LIN {X -0.161,Y -632.553,Z 539.342,A 0.000,B 0.000,C 90.000,E1 97.587} C_DIS
LIN {X 0.137,Y -636.870,Z 539.336,A 0.000,B 0.000,C 90.000,E1 96.549} C_DIS
LIN {X 0.117,Y -640.044,Z 539.332,A 0.000,B 0.000,C 90.000,E1 95.796} C_DIS
LIN {X -0.184,Y -643.748,Z 539.327,A 0.000,B 0.000,C 90.000,E1 94.821} C_DIS
LIN {X -0.199,Y -646.261,Z 539.323,A 0.000,B 0.000,C 90.000,E1 94.073} C_DIS
LIN {X -0.191,Y -648.527,Z 539.318,A 0.000,B 0.000,C 90.000,E1 93.326} C_DIS
LIN {X -0.164,Y -650.528,Z 539.314,A 0.000,B 0.000,C 90.000,E1 92.579} C_DIS
LIN {X -0.144,Y -652.163,Z 539.310,A 0.000,B 0.000,C 90.000,E1 91.835} C_DIS
LIN {X -0.091,Y -653.365,Z 539.306,A 0.000,B 0.000,C 90.000,E1 91.088} C_DIS
LIN {X 0.160,Y -654.029,Z 539.303,A 0.000,B 0.000,C 90.000,E1 90.573} C_DIS
LIN {X -0.239,Y -654.516,Z 539.301,A 0.000,B 0.000,C 90.000,E1 90.115} C_DIS
LIN {X -0.177,Y -654.885,Z 539.296,A 0.000,B 0.000,C 90.000,E1 89.370} C_DIS
LIN {X 0.085,Y -654.983,Z 539.294,A 0.000,B 0.000,C 90.000,E1 88.854} C_DIS
LIN {X 0.168,Y -654.825,Z 539.290,A 0.000,B 0.000,C 90.000,E1 88.108} C_DIS
LIN {X -0.226,Y -654.541,Z 539.287,A 0.000,B 0.000,C 90.000,E1 87.650} C_DIS
LIN {X -0.173,Y -653.859,Z 539.283,A 0.000,B 0.000,C 90.000,E1 86.906} C_DIS
LIN {X -0.257,Y -652.473,Z 539.277,A 0.000,B 0.000,C 90.000,E1 85.927} C_DIS
LIN {X 0.186,Y -652.109,Z 539.276,A 0.000,B 0.000,C 90.000,E1 85.641} C_DIS
LIN {X -0.127,Y -649.508,Z 539.269,A 0.000,B 0.000,C 90.000,E1 84.432} C_DIS
LIN {X 0.138,Y -648.367,Z 539.266,A 0.000,B 0.000,C 90.000,E1 83.913} C_DIS
LIN {X 0.000,Y -645.573,Z 539.261,A 0.000,B 0.000,C 90.000,E1 82.932} C_DIS
LIN {X 0.237,Y -643.951,Z 539.258,A 0.000,B 0.000,C 90.000,E1 82.413} C_DIS
LIN {X 0.034,Y -640.529,Z 539.252,A 0.000,B 0.000,C 90.000,E1 81.432} C_DIS
LIN {X 0.227,Y -638.679,Z 539.250,A 0.000,B 0.000,C 90.000,E1 80.914} C_DIS
LIN {X 0.333,Y -635.655,Z 539.245,A 0.000,B 0.000,C 90.000,E1 80.151} C_DIS
LIN {X -0.136,Y -633.425,Z 539.243,A 0.000,B 0.000,C 90.000,E1 79.690} C_DIS
LIN {X -0.226,Y -629.355,Z 539.238,A 0.000,B 0.000,C 90.000,E1 78.814} C_DIS
LIN {X -0.190,Y -625.693,Z 539.234,A 0.000,B 0.000,C 90.000,E1 78.049} C_DIS
LIN {X -0.215,Y -619.808,Z 539.227,A 0.000,B 0.000,C 90.000,E1 76.937} C_DIS
LIN {X -0.057,Y -616.886,Z 539.224,A 0.000,B 0.000,C 90.000,E1 76.408} C_DIS
LIN {X -0.161,Y -612.053,Z 539.220,A 0.000,B 0.000,C 90.000,E1 75.644} C_DIS
LIN {X 0.217,Y -605.780,Z 539.215,A 0.000,B 0.000,C 90.000,E1 74.700} C_DIS
LIN {X 0.209,Y -600.730,Z 539.212,A 0.000,B 0.000,C 90.000,E1 74.047} C_DIS
LIN {X -0.187,Y -596.279,Z 539.209,A 0.000,B 0.000,C 90.000,E1 73.559} C_DIS
LIN {X -0.213,Y -590.050,Z 539.205,A 0.000,B 0.000,C 90.000,E1 72.906} C_DIS
LIN {X 0.120,Y -586.238,Z 539.203,A 0.000,B 0.000,C 90.000,E1 72.489} C_DIS
LIN {X 0.255,Y -580.969,Z 539.200,A 0.000,B 0.000,C 90.000,E1 72.000} C_DIS
LIN {X -0.331,Y -573.128,Z 539.197,A 0.000,B 0.000,C 90.000,E1 71.402} C_DIS
LIN {X -0.139,Y -568.567,Z 539.195,A 0.000,B 0.000,C 90.000,E1 71.040} C_DIS
LIN {X 0.221,Y -563.998,Z 539.193,A 0.000,B 0.000,C 90.000,E1 70.678} C_DIS
LIN {X -0.057,Y -557.456,Z 539.191,A 0.000,B 0.000,C 90.000,E1 70.296} C_DIS
LIN {X 0.145,Y -549.435,Z 539.188,A 0.000,B 0.000,C 90.000,E1 69.826} C_DIS
LIN {X -0.129,Y -542.518,Z 539.186,A 0.000,B 0.000,C 90.000,E1 69.518} C_DIS
LIN {X -0.088,Y -535.231,Z 539.185,A 0.000,B 0.000,C 90.000,E1 69.209} C_DIS
LIN {X -0.199,Y -527.996,Z 539.183,A 0.000,B 0.000,C 90.000,E1 68.954} C_DIS
LIN {X -0.211,Y -517.329,Z 539.181,A 0.000,B 0.000,C 90.000,E1 68.592} C_DIS
LIN {X 0.274,Y -504.903,Z 539.179,A 0.000,B 0.000,C 90.000,E1 68.156} C_DIS
LIN {X -0.019,Y -497.455,Z 539.178,A 0.000,B 0.000,C 90.000,E1 67.975} C_DIS
LIN {X 0.175,Y -485.004,Z 539.176,A 0.000,B 0.000,C 90.000,E1 67.614} C_DIS
LIN {X 0.015,Y -465.783,Z 539.173,A 0.000,B 0.000,C 90.000,E1 67.102} C_DIS
LIN {X -0.011,Y -465.706,Z 539.173,A 0.000,B 0.000,C 90.000,E1 67.102} C_DIS
LIN {X -0.282,Y -455.953,Z 539.146,A 0.000,B 0.000,C 90.000,E1 62.231} C_DIS
LIN {X -0.176,Y -455.427,Z 539.144,A 0.000,B 0.000,C 90.000,E1 61.897} C_DIS
LIN {X 0.140,Y -446.089,Z 539.120,A 0.000,B 0.000,C 90.000,E1 57.661} C_DIS
LIN {X 0.017,Y -443.661,Z 539.113,A 0.000,B 0.000,C 90.000,E1 56.373} C_DIS
LIN {X 0.047,Y -443.048,Z 539.112,A 0.000,B 0.000,C 90.000,E1 56.135} C_DIS
LIN {X 0.007,Y -443.048,Z 539.112,A 0.000,B 0.000,C 90.000,E1 56.135} C_DIS
LIN {X 0.110,Y -446.646,Z 539.102,A 0.000,B 0.000,C 90.000,E1 54.402} C_DIS
LIN {X 0.221,Y -449.820,Z 539.093,A 0.000,B 0.000,C 90.000,E1 52.763} C_DIS
LIN {X 0.040,Y -452.125,Z 539.086,A 0.000,B 0.000,C 90.000,E1 51.492} C_DIS
LIN {X 0.099,Y -453.720,Z 539.081,A 0.000,B 0.000,C 90.000,E1 50.517} C_DIS
LIN {X 0.196,Y -455.801,Z 539.074,A 0.000,B 0.000,C 90.000,E1 49.218} C_DIS
LIN {X 0.025,Y -457.655,Z 539.066,A 0.000,B 0.000,C 90.000,E1 47.957} C_DIS
LIN {X -0.158,Y -459.271,Z 539.059,A 0.000,B 0.000,C 90.000,E1 46.701} C_DIS
LIN {X 0.003,Y -460.455,Z 539.052,A 0.000,B 0.000,C 90.000,E1 45.405} C_DIS
LIN {X 0.140,Y -461.157,Z 539.047,A 0.000,B 0.000,C 90.000,E1 44.433} C_DIS
LIN {X -0.036,Y -461.732,Z 539.042,A 0.000,B 0.000,C 90.000,E1 43.500} C_DIS
LIN {X 0.160,Y -462.205,Z 539.035,A 0.000,B 0.000,C 90.000,E1 42.204} C_DIS
LIN {X 0.083,Y -462.454,Z 539.028,A 0.000,B 0.000,C 90.000,E1 40.943} C_DIS
LIN {X -0.039,Y -462.485,Z 539.021,A 0.000,B 0.000,C 90.000,E1 39.688} C_DIS
LIN {X 0.248,Y -462.250,Z 539.013,A 0.000,B 0.000,C 90.000,E1 38.382} C_DIS
LIN {X 0.141,Y -461.964,Z 539.008,A 0.000,B 0.000,C 90.000,E1 37.443} C_DIS
LIN {X -0.104,Y -461.385,Z 538.999,A 0.000,B 0.000,C 90.000,E1 35.884} C_DIS
LIN {X -0.117,Y -460.356,Z 538.987,A 0.000,B 0.000,C 90.000,E1 33.658} C_DIS
LIN {X -0.026,Y -459.616,Z 538.978,A 0.000,B 0.000,C 90.000,E1 32.054} C_DIS
LIN {X -0.055,Y -458.897,Z 538.969,A 0.000,B 0.000,C 90.000,E1 30.463} C_DIS
LIN {X -0.200,Y -457.939,Z 538.959,A 0.000,B 0.000,C 90.000,E1 28.565} C_DIS
LIN {X -0.071,Y -457.170,Z 538.950,A 0.000,B 0.000,C 90.000,E1 26.950} C_DIS
LIN {X 0.032,Y -456.139,Z 538.937,A 0.000,B 0.000,C 90.000,E1 24.695} C_DIS
LIN {X -0.155,Y -455.183,Z 538.923,A 0.000,B 0.000,C 90.000,E1 22.153} C_DIS
LIN {X 0.100,Y -454.615,Z 538.912,A 0.000,B 0.000,C 90.000,E1 20.194} C_DIS
LIN {X 0.012,Y -454.238,Z 538.903,A 0.000,B 0.000,C 90.000,E1 18.598} C_DIS
LIN {X 0.057,Y -454.011,Z 538.894,A 0.000,B 0.000,C 90.000,E1 16.985} C_DIS
LIN {X -0.179,Y -453.989,Z 538.878,A 0.000,B 0.000,C 90.000,E1 14.120} C_DIS
LIN {X -0.102,Y -454.567,Z 538.860,A 0.000,B 0.000,C 90.000,E1 10.894} C_DIS
LIN {X -0.233,Y -455.490,Z 538.846,A 0.000,B 0.000,C 90.000,E1 8.341} C_DIS
LIN {X -0.165,Y -456.606,Z 538.834,A 0.000,B 0.000,C 90.000,E1 6.087} C_DIS
LIN {X 0.061,Y -458.239,Z 538.820,A 0.000,B 0.000,C 90.000,E1 3.498} C_DIS
LIN {X 0.078,Y -459.999,Z 538.807,A 0.000,B 0.000,C 90.000,E1 1.260} C_DIS
LIN {X -0.172,Y -463.198,Z 538.790,A 0.000,B 0.000,C 90.000,E1 358.224} C_DIS
LIN {X -0.016,Y -466.734,Z 538.774,A 0.000,B 0.000,C 90.000,E1 355.355} C_DIS
LIN {X 0.090,Y -469.208,Z 538.764,A 0.000,B 0.000,C 90.000,E1 353.451} C_DIS
LIN {X 0.085,Y -472.158,Z 538.752,A 0.000,B 0.000,C 90.000,E1 351.254} C_DIS
LIN {X 0.220,Y -475.229,Z 538.739,A 0.000,B 0.000,C 90.000,E1 349.050} C_DIS
LIN {X -0.047,Y -479.727,Z 538.724,A 0.000,B 0.000,C 90.000,E1 346.284} C_DIS
LIN {X 0.102,Y -484.216,Z 538.710,A 0.000,B 0.000,C 90.000,E1 343.795} C_DIS
LIN {X 0.036,Y -488.962,Z 538.696,A 0.000,B 0.000,C 90.000,E1 341.348} C_DIS
LIN {X 0.038,Y -492.574,Z 538.686,A 0.000,B 0.000,C 90.000,E1 339.518} C_DIS
LIN {X -0.102,Y -496.765,Z 538.674,A 0.000,B 0.000,C 90.000,E1 337.411} C_DIS
LIN {X -0.204,Y -500.238,Z 538.664,A 0.000,B 0.000,C 90.000,E1 335.613} C_DIS
LIN {X -0.180,Y -502.462,Z 538.658,A 0.000,B 0.000,C 90.000,E1 334.409} C_DIS
LIN {X -0.195,Y -505.759,Z 538.648,A 0.000,B 0.000,C 90.000,E1 332.615} C_DIS
LIN {X 0.096,Y -508.923,Z 538.638,A 0.000,B 0.000,C 90.000,E1 330.795} C_DIS
LIN {X 0.269,Y -512.153,Z 538.628,A 0.000,B 0.000,C 90.000,E1 328.997} C_DIS
LIN {X 0.077,Y -515.372,Z 538.618,A 0.000,B 0.000,C 90.000,E1 327.248} C_DIS
LIN {X -0.135,Y -518.119,Z 538.610,A 0.000,B 0.000,C 90.000,E1 325.801} C_DIS
LIN {X -0.001,Y -520.822,Z 538.602,A 0.000,B 0.000,C 90.000,E1 324.322} C_DIS
LIN {X 0.141,Y -524.009,Z 538.592,A 0.000,B 0.000,C 90.000,E1 322.557} C_DIS
LIN {X 0.251,Y -527.316,Z 538.582,A 0.000,B 0.000,C 90.000,E1 320.803} C_DIS
LIN {X -0.116,Y -533.148,Z 538.566,A 0.000,B 0.000,C 90.000,E1 317.957} C_DIS
LIN {X -0.315,Y -537.519,Z 538.555,A 0.000,B 0.000,C 90.000,E1 315.972} C_DIS
LIN {X -0.022,Y -543.522,Z 538.541,A 0.000,B 0.000,C 90.000,E1 313.380} C_DIS
LIN {X 0.027,Y -546.374,Z 538.535,A 0.000,B 0.000,C 90.000,E1 312.243} C_DIS
LIN {X -0.288,Y -549.138,Z 538.529,A 0.000,B 0.000,C 90.000,E1 311.148} C_DIS
LIN {X 0.213,Y -551.048,Z 538.524,A 0.000,B 0.000,C 90.000,E1 310.253} C_DIS
LIN {X 0.008,Y -554.086,Z 538.516,A 0.000,B 0.000,C 90.000,E1 308.874} C_DIS
LIN {X 0.369,Y -557.334,Z 538.508,A 0.000,B 0.000,C 90.000,E1 307.443} C_DIS
LIN {X -0.248,Y -558.907,Z 538.505,A 0.000,B 0.000,C 90.000,E1 306.950} C_DIS
LIN {X -0.037,Y -559.427,Z 538.504,A 0.000,B 0.000,C 90.000,E1 306.790} C_DIS
LIN {X -0.070,Y -561.428,Z 538.502,A 0.000,B 0.000,C 90.000,E1 306.377} C_DIS
LIN {X 0.026,Y -563.355,Z 538.501,A 0.000,B 0.000,C 90.000,E1 306.091} C_DIS
LIN {X 0.129,Y -565.266,Z 538.499,A 0.000,B 0.000,C 90.000,E1 305.804} C_DIS
LIN {X 0.149,Y -568.092,Z 538.497,A 0.000,B 0.000,C 90.000,E1 305.438} C_DIS
LIN {X 0.008,Y -570.735,Z 538.496,A 0.000,B 0.000,C 90.000,E1 305.185} C_DIS
LIN {X 0.208,Y -572.950,Z 538.494,A 0.000,B 0.000,C 90.000,E1 304.898} C_DIS
LIN {X 0.069,Y -576.395,Z 538.492,A 0.000,B 0.000,C 90.000,E1 304.565} C_DIS
LIN {X -0.134,Y -578.700,Z 538.491,A 0.000,B 0.000,C 90.000,E1 304.326} C_DIS
LIN {X -0.132,Y -585.903,Z 538.487,A 0.000,B 0.000,C 90.000,E1 303.579} C_DIS
LIN {X 0.109,Y -591.873,Z 538.483,A 0.000,B 0.000,C 90.000,E1 302.911} C_DIS
LIN {X -0.130,Y -602.582,Z 538.476,A 0.000,B 0.000,C 90.000,E1 301.750} C_DIS
LIN {X 0.293,Y -609.452,Z 538.472,A 0.000,B 0.000,C 90.000,E1 300.924} C_DIS
LIN {X -0.349,Y -614.898,Z 538.468,A 0.000,B 0.000,C 90.000,E1 300.335} C_DIS
LIN {X -0.098,Y -618.893,Z 538.466,A 0.000,B 0.000,C 90.000,E1 299.795} C_DIS
LIN {X -0.125,Y -622.479,Z 538.463,A 0.000,B 0.000,C 90.000,E1 299.283} C_DIS
LIN {X 0.177,Y -625.745,Z 538.460,A 0.000,B 0.000,C 90.000,E1 298.743} C_DIS
LIN {X 0.192,Y -627.757,Z 538.458,A 0.000,B 0.000,C 90.000,E1 298.359} C_DIS
LIN {X 0.231,Y -629.993,Z 538.455,A 0.000,B 0.000,C 90.000,E1 297.847} C_DIS
LIN {X -0.304,Y -630.974,Z 538.453,A 0.000,B 0.000,C 90.000,E1 297.641} C_DIS
LIN {X -0.277,Y -631.817,Z 538.452,A 0.000,B 0.000,C 90.000,E1 297.385} C_DIS
LIN {X -0.212,Y -633.149,Z 538.449,A 0.000,B 0.000,C 90.000,E1 296.873} C_DIS
LIN {X -0.136,Y -633.784,Z 538.446,A 0.000,B 0.000,C 90.000,E1 296.360} C_DIS
LIN {X -0.096,Y -634.016,Z 538.445,A 0.000,B 0.000,C 90.000,E1 296.104} C_DIS
LIN {X -0.015,Y -633.509,Z 538.442,A 0.000,B 0.000,C 90.000,E1 295.591} C_DIS
LIN {X 0.025,Y -633.147,Z 538.441,A 0.000,B 0.000,C 90.000,E1 295.335} C_DIS
LIN {X 0.063,Y -632.018,Z 538.439,A 0.000,B 0.000,C 90.000,E1 295.079} C_DIS
LIN {X 0.100,Y -631.238,Z 538.438,A 0.000,B 0.000,C 90.000,E1 294.823} C_DIS
LIN {X -0.148,Y -630.640,Z 538.437,A 0.000,B 0.000,C 90.000,E1 294.719} C_DIS
LIN {X -0.116,Y -629.010,Z 538.436,A 0.000,B 0.000,C 90.000,E1 294.463} C_DIS
LIN {X -0.102,Y -628.001,Z 538.435,A 0.000,B 0.000,C 90.000,E1 294.335} C_DIS
LIN {X -0.079,Y -625.339,Z 538.434,A 0.000,B 0.000,C 90.000,E1 294.079} C_DIS
LIN {X -0.049,Y -622.387,Z 538.433,A 0.000,B 0.000,C 90.000,E1 293.898} C_DIS
LIN {X 0.191,Y -620.518,Z 538.432,A 0.000,B 0.000,C 90.000,E1 293.695} C_DIS
LIN {X 0.007,Y -618.872,Z 538.431,A 0.000,B 0.000,C 90.000,E1 293.590} C_DIS
LIN {X 0.043,Y -611.966,Z 538.429,A 0.000,B 0.000,C 90.000,E1 293.206} C_DIS
LIN {X -0.106,Y -602.994,Z 538.427,A 0.000,B 0.000,C 90.000,E1 292.823} C_DIS
LIN {X 0.327,Y -596.063,Z 538.425,A 0.000,B 0.000,C 90.000,E1 292.514} C_DIS
LIN {X -0.216,Y -590.775,Z 538.424,A 0.000,B 0.000,C 90.000,E1 292.386} C_DIS
LIN {X -0.212,Y -583.096,Z 538.423,A 0.000,B 0.000,C 90.000,E1 292.078} C_DIS
LIN {X -0.184,Y -578.414,Z 538.421,A 0.000,B 0.000,C 90.000,E1 291.844} C_DIS
LIN {X 0.056,Y -576.702,Z 538.421,A 0.000,B 0.000,C 90.000,E1 291.716} C_DIS
LIN {X -0.083,Y -574.112,Z 538.420,A 0.000,B 0.000,C 90.000,E1 291.535} C_DIS
LIN {X -0.029,Y -573.253,Z 538.419,A 0.000,B 0.000,C 90.000,E1 291.408} C_DIS
LIN {X 0.063,Y -572.549,Z 538.417,A 0.000,B 0.000,C 90.000,E1 291.099} C_DIS
LIN {X -0.328,Y -572.335,Z 538.413,A 0.000,B 0.000,C 90.000,E1 290.429} C_DIS
LIN {X 0.013,Y -572.469,Z 538.409,A 0.000,B 0.000,C 90.000,E1 289.577} C_DIS
LIN {X -0.200,Y -572.511,Z 538.401,A 0.000,B 0.000,C 90.000,E1 288.236} C_DIS
LIN {X -0.053,Y -572.295,Z 538.394,A 0.000,B 0.000,C 90.000,E1 286.858} C_DIS
LIN {X -0.251,Y -571.983,Z 538.388,A 0.000,B 0.000,C 90.000,E1 285.788} C_DIS
LIN {X 0.068,Y -571.227,Z 538.379,A 0.000,B 0.000,C 90.000,E1 284.120} C_DIS
LIN {X 0.091,Y -570.432,Z 538.369,A 0.000,B 0.000,C 90.000,E1 282.479} C_DIS
LIN {X 0.105,Y -569.643,Z 538.360,A 0.000,B 0.000,C 90.000,E1 280.838} C_DIS
LIN {X 0.283,Y -569.045,Z 538.354,A 0.000,B 0.000,C 90.000,E1 279.726} C_DIS
LIN {X 0.059,Y -568.241,Z 538.345,A 0.000,B 0.000,C 90.000,E1 278.106} C_DIS
LIN {X -0.181,Y -567.557,Z 538.336,A 0.000,B 0.000,C 90.000,E1 276.486} C_DIS
LIN {X -0.209,Y -567.219,Z 538.330,A 0.000,B 0.000,C 90.000,E1 275.391} C_DIS
LIN {X 0.165,Y -566.883,Z 538.325,A 0.000,B 0.000,C 90.000,E1 274.531} C_DIS
LIN {X 0.087,Y -566.382,Z 538.319,A 0.000,B 0.000,C 90.000,E1 273.440} C_DIS
LIN {X 0.248,Y -565.415,Z 538.310,A 0.000,B 0.000,C 90.000,E1 271.776} C_DIS
LIN {X 0.129,Y -564.763,Z 538.304,A 0.000,B 0.000,C 90.000,E1 270.688} C_DIS
LIN {X 0.221,Y -563.529,Z 538.295,A 0.000,B 0.000,C 90.000,E1 269.026} C_DIS
LIN {X 0.196,Y -562.554,Z 538.287,A 0.000,B 0.000,C 90.000,E1 267.650} C_DIS
LIN {X -0.092,Y -561.020,Z 538.275,A 0.000,B 0.000,C 90.000,E1 265.469} C_DIS
LIN {X -0.209,Y -560.118,Z 538.269,A 0.000,B 0.000,C 90.000,E1 264.375} C_DIS
LIN {X -0.197,Y -558.958,Z 538.261,A 0.000,B 0.000,C 90.000,E1 262.989} C_DIS
LIN {X -0.150,Y -557.527,Z 538.252,A 0.000,B 0.000,C 90.000,E1 261.319} C_DIS
LIN {X 0.123,Y -556.936,Z 538.249,A 0.000,B 0.000,C 90.000,E1 260.735} C_DIS
LIN {X -0.134,Y -554.565,Z 538.238,A 0.000,B 0.000,C 90.000,E1 258.814} C_DIS
LIN {X -0.167,Y -553.164,Z 538.232,A 0.000,B 0.000,C 90.000,E1 257.701} C_DIS
LIN {X -0.223,Y -551.701,Z 538.225,A 0.000,B 0.000,C 90.000,E1 256.589} C_DIS
LIN {X -0.173,Y -550.104,Z 538.219,A 0.000,B 0.000,C 90.000,E1 255.463} C_DIS
LIN {X 0.102,Y -547.909,Z 538.211,A 0.000,B 0.000,C 90.000,E1 254.031} C_DIS
LIN {X -0.182,Y -545.529,Z 538.204,A 0.000,B 0.000,C 90.000,E1 252.653} C_DIS
LIN {X -0.062,Y -543.444,Z 538.197,A 0.000,B 0.000,C 90.000,E1 251.511} C_DIS
LIN {X 0.019,Y -541.277,Z 538.191,A 0.000,B 0.000,C 90.000,E1 250.369} C_DIS
LIN {X 0.018,Y -539.529,Z 538.186,A 0.000,B 0.000,C 90.000,E1 249.518} C_DIS
LIN {X -0.069,Y -536.536,Z 538.178,A 0.000,B 0.000,C 90.000,E1 248.103} C_DIS
LIN {X 0.282,Y -533.977,Z 538.172,A 0.000,B 0.000,C 90.000,E1 246.922} C_DIS
LIN {X 0.106,Y -531.238,Z 538.166,A 0.000,B 0.000,C 90.000,E1 245.793} C_DIS
LIN {X -0.109,Y -528.344,Z 538.159,A 0.000,B 0.000,C 90.000,E1 244.665} C_DIS
LIN {X -0.141,Y -525.295,Z 538.153,A 0.000,B 0.000,C 90.000,E1 243.512} C_DIS
LIN {X 0.172,Y -521.296,Z 538.145,A 0.000,B 0.000,C 90.000,E1 242.025} C_DIS
LIN {X -0.049,Y -517.287,Z 538.137,A 0.000,B 0.000,C 90.000,E1 240.589} C_DIS
LIN {X 0.000,Y -513.994,Z 538.130,A 0.000,B 0.000,C 90.000,E1 239.410} C_DIS
LIN {X 0.257,Y -510.493,Z 538.124,A 0.000,B 0.000,C 90.000,E1 238.201} C_DIS
LIN {X 0.251,Y -505.166,Z 538.114,A 0.000,B 0.000,C 90.000,E1 236.421} C_DIS
LIN {X -0.002,Y -498.995,Z 538.102,A 0.000,B 0.000,C 90.000,E1 234.356} C_DIS
LIN {X -0.094,Y -493.882,Z 538.092,A 0.000,B 0.000,C 90.000,E1 232.557} C_DIS
LIN {X 0.163,Y -491.395,Z 538.087,A 0.000,B 0.000,C 90.000,E1 231.618} C_DIS
LIN {X -0.202,Y -484.785,Z 538.073,A 0.000,B 0.000,C 90.000,E1 229.218} C_DIS
LIN {X 0.318,Y -479.992,Z 538.063,A 0.000,B 0.000,C 90.000,E1 227.310} C_DIS
LIN {X 0.125,Y -474.601,Z 538.051,A 0.000,B 0.000,C 90.000,E1 225.162} C_DIS
LIN {X 0.034,Y -470.009,Z 538.041,A 0.000,B 0.000,C 90.000,E1 223.299} C_DIS
LIN {X -0.211,Y -466.360,Z 538.032,A 0.000,B 0.000,C 90.000,E1 221.757} C_DIS
LIN {X -0.172,Y -462.733,Z 538.023,A 0.000,B 0.000,C 90.000,E1 220.172} C_DIS
LIN {X -0.108,Y -458.490,Z 538.013,A 0.000,B 0.000,C 90.000,E1 218.257} C_DIS
LIN {X 0.213,Y -454.346,Z 538.002,A 0.000,B 0.000,C 90.000,E1 216.297} C_DIS
LIN {X -0.020,Y -449.641,Z 537.989,A 0.000,B 0.000,C 90.000,E1 214.072} C_DIS
LIN {X -0.074,Y -445.754,Z 537.979,A 0.000,B 0.000,C 90.000,E1 212.133} C_DIS
LIN {X 0.237,Y -442.641,Z 537.969,A 0.000,B 0.000,C 90.000,E1 210.463} C_DIS
LIN {X -0.252,Y -438.429,Z 537.957,A 0.000,B 0.000,C 90.000,E1 208.231} C_DIS
LIN {X -0.086,Y -434.500,Z 537.944,A 0.000,B 0.000,C 90.000,E1 205.899} C_DIS
LIN {X -0.027,Y -430.698,Z 537.931,A 0.000,B 0.000,C 90.000,E1 203.567} C_DIS
LIN {X -0.009,Y -427.128,Z 537.918,A 0.000,B 0.000,C 90.000,E1 201.227} C_DIS
LIN {X 0.143,Y -423.016,Z 537.901,A 0.000,B 0.000,C 90.000,E1 198.181} C_DIS
LIN {X -0.235,Y -420.439,Z 537.890,A 0.000,B 0.000,C 90.000,E1 196.205} C_DIS
LIN {X -0.026,Y -418.448,Z 537.880,A 0.000,B 0.000,C 90.000,E1 194.481} C_DIS
LIN {X -0.015,Y -416.769,Z 537.873,A 0.000,B 0.000,C 90.000,E1 193.119} C_DIS
LIN {X -0.081,Y -414.634,Z 537.863,A 0.000,B 0.000,C 90.000,E1 191.422} C_DIS
LIN {X 0.216,Y -412.659,Z 537.854,A 0.000,B 0.000,C 90.000,E1 189.670} C_DIS
LIN {X -0.040,Y -410.381,Z 537.842,A 0.000,B 0.000,C 90.000,E1 187.644} C_DIS
LIN {X 0.025,Y -407.915,Z 537.829,A 0.000,B 0.000,C 90.000,E1 185.220} C_DIS
LIN {X -0.056,Y -405.786,Z 537.816,A 0.000,B 0.000,C 90.000,E1 182.808} C_DIS
LIN {X 0.111,Y -403.421,Z 537.798,A 0.000,B 0.000,C 90.000,E1 179.656} C_DIS
LIN {X -0.166,Y -402.020,Z 537.783,A 0.000,B 0.000,C 90.000,E1 176.906} C_DIS
LIN {X -0.021,Y -401.143,Z 537.767,A 0.000,B 0.000,C 90.000,E1 174.090} C_DIS
LIN {X -0.147,Y -400.760,Z 537.754,A 0.000,B 0.000,C 90.000,E1 171.659} C_DIS
LIN {X 0.193,Y -400.781,Z 537.742,A 0.000,B 0.000,C 90.000,E1 169.511} C_DIS
LIN {X 0.219,Y -400.966,Z 537.732,A 0.000,B 0.000,C 90.000,E1 167.757} C_DIS
LIN {X -0.005,Y -401.545,Z 537.717,A 0.000,B 0.000,C 90.000,E1 164.991} C_DIS
LIN {X -0.084,Y -402.293,Z 537.705,A 0.000,B 0.000,C 90.000,E1 162.906} C_DIS
LIN {X 0.100,Y -403.197,Z 537.693,A 0.000,B 0.000,C 90.000,E1 160.786} C_DIS
LIN {X -0.073,Y -404.315,Z 537.682,A 0.000,B 0.000,C 90.000,E1 158.720} C_DIS
LIN {X 0.067,Y -405.521,Z 537.670,A 0.000,B 0.000,C 90.000,E1 156.613} C_DIS
LIN {X 0.028,Y -406.879,Z 537.659,A 0.000,B 0.000,C 90.000,E1 154.537} C_DIS
LIN {X 0.105,Y -408.087,Z 537.649,A 0.000,B 0.000,C 90.000,E1 152.794} C_DIS
LIN {X 0.210,Y -409.252,Z 537.639,A 0.000,B 0.000,C 90.000,E1 151.051} C_DIS
LIN {X 0.250,Y -410.059,Z 537.632,A 0.000,B 0.000,C 90.000,E1 149.665} C_DIS
LIN {X -0.123,Y -410.903,Z 537.622,A 0.000,B 0.000,C 90.000,E1 147.995} C_DIS
LIN {X -0.267,Y -411.684,Z 537.613,A 0.000,B 0.000,C 90.000,E1 146.294} C_DIS
LIN {X -0.171,Y -412.256,Z 537.603,A 0.000,B 0.000,C 90.000,E1 144.562} C_DIS
LIN {X -0.160,Y -412.731,Z 537.594,A 0.000,B 0.000,C 90.000,E1 142.844} C_DIS
LIN {X 0.117,Y -413.084,Z 537.584,A 0.000,B 0.000,C 90.000,E1 141.090} C_DIS
LIN {X -0.062,Y -413.413,Z 537.573,A 0.000,B 0.000,C 90.000,E1 139.057} C_DIS
LIN {X 0.039,Y -413.513,Z 537.561,A 0.000,B 0.000,C 90.000,E1 136.986} C_DIS
LIN {X 0.115,Y -413.573,Z 537.550,A 0.000,B 0.000,C 90.000,E1 134.919} C_DIS
LIN {X 0.163,Y -413.623,Z 537.542,A 0.000,B 0.000,C 90.000,E1 133.542} C_DIS
LIN {X 0.091,Y -413.600,Z 537.533,A 0.000,B 0.000,C 90.000,E1 131.838} C_DIS
LIN {X 0.156,Y -413.295,Z 537.525,A 0.000,B 0.000,C 90.000,E1 130.458} C_DIS
LIN {X 0.092,Y -412.975,Z 537.519,A 0.000,B 0.000,C 90.000,E1 129.439} C_DIS
LIN {X 0.046,Y -412.077,Z 537.510,A 0.000,B 0.000,C 90.000,E1 127.729} C_DIS
LIN {X -0.078,Y -411.776,Z 537.507,A 0.000,B 0.000,C 90.000,E1 127.237} C_DIS
LIN {X -0.117,Y -411.774,Z 537.507,A 0.000,B 0.000,C 90.000,E1 127.237} C_DIS
LIN {X 0.058,Y -415.387,Z 537.500,A 0.000,B 0.000,C 90.000,E1 126.011} C_DIS
LIN {X 0.120,Y -425.790,Z 537.478,A 0.000,B 0.000,C 90.000,E1 121.926} C_DIS
LIN {X 0.064,Y -430.822,Z 537.468,A 0.000,B 0.000,C 90.000,E1 120.256} C_DIS
LIN {X 0.024,Y -440.786,Z 537.446,A 0.000,B 0.000,C 90.000,E1 116.283} C_DIS
LIN {X -0.007,Y -444.653,Z 537.439,A 0.000,B 0.000,C 90.000,E1 114.975} C_DIS
LIN {X -0.030,Y -447.709,Z 537.431,A 0.000,B 0.000,C 90.000,E1 113.567} C_DIS
LIN {X -0.069,Y -447.773,Z 537.431,A 0.000,B 0.000,C 90.000,E1 113.567} C_DIS
LIN {X 0.122,Y -479.243,Z 537.424,A 0.000,B 0.000,C 90.000,E1 112.280} C_DIS
LIN {X -0.156,Y -487.869,Z 537.422,A 0.000,B 0.000,C 90.000,E1 111.972} C_DIS
LIN {X 0.153,Y -503.313,Z 537.418,A 0.000,B 0.000,C 90.000,E1 111.280} C_DIS
LIN {X 0.061,Y -511.784,Z 537.416,A 0.000,B 0.000,C 90.000,E1 110.918} C_DIS
LIN {X -0.130,Y -521.990,Z 537.414,A 0.000,B 0.000,C 90.000,E1 110.482} C_DIS
LIN {X -0.059,Y -531.923,Z 537.411,A 0.000,B 0.000,C 90.000,E1 109.993} C_DIS
LIN {X 0.202,Y -538.437,Z 537.409,A 0.000,B 0.000,C 90.000,E1 109.631} C_DIS
LIN {X -0.196,Y -544.767,Z 537.407,A 0.000,B 0.000,C 90.000,E1 109.322} C_DIS
LIN {X -0.088,Y -549.449,Z 537.406,A 0.000,B 0.000,C 90.000,E1 109.033} C_DIS
LIN {X 0.282,Y -555.650,Z 537.404,A 0.000,B 0.000,C 90.000,E1 108.598} C_DIS
LIN {X 0.149,Y -561.521,Z 537.401,A 0.000,B 0.000,C 90.000,E1 108.181} C_DIS
LIN {X -0.267,Y -567.094,Z 537.399,A 0.000,B 0.000,C 90.000,E1 107.764} C_DIS
LIN {X -0.266,Y -572.433,Z 537.396,A 0.000,B 0.000,C 90.000,E1 107.275} C_DIS
LIN {X 0.039,Y -577.565,Z 537.393,A 0.000,B 0.000,C 90.000,E1 106.732} C_DIS
LIN {X -0.132,Y -583.440,Z 537.389,A 0.000,B 0.000,C 90.000,E1 106.079} C_DIS
LIN {X 0.250,Y -588.910,Z 537.386,A 0.000,B 0.000,C 90.000,E1 105.371} C_DIS
LIN {X 0.344,Y -592.865,Z 537.383,A 0.000,B 0.000,C 90.000,E1 104.828} C_DIS
LIN {X 0.090,Y -597.387,Z 537.379,A 0.000,B 0.000,C 90.000,E1 104.189} C_DIS
LIN {X -0.292,Y -601.563,Z 537.375,A 0.000,B 0.000,C 90.000,E1 103.592} C_DIS
LIN {X 0.057,Y -606.543,Z 537.371,A 0.000,B 0.000,C 90.000,E1 102.771} C_DIS
LIN {X 0.059,Y -610.570,Z 537.367,A 0.000,B 0.000,C 90.000,E1 102.119} C_DIS
LIN {X -0.281,Y -615.771,Z 537.362,A 0.000,B 0.000,C 90.000,E1 101.243} C_DIS
LIN {X 0.278,Y -619.182,Z 537.359,A 0.000,B 0.000,C 90.000,E1 100.546} C_DIS
LIN {X -0.184,Y -621.704,Z 537.356,A 0.000,B 0.000,C 90.000,E1 100.074} C_DIS
LIN {X -0.268,Y -627.612,Z 537.349,A 0.000,B 0.000,C 90.000,E1 98.803} C_DIS
LIN {X -0.245,Y -633.134,Z 537.342,A 0.000,B 0.000,C 90.000,E1 97.530} C_DIS
LIN {X 0.135,Y -637.513,Z 537.336,A 0.000,B 0.000,C 90.000,E1 96.486} C_DIS
LIN {X 0.050,Y -640.699,Z 537.332,A 0.000,B 0.000,C 90.000,E1 95.739} C_DIS
LIN {X -0.188,Y -644.435,Z 537.326,A 0.000,B 0.000,C 90.000,E1 94.759} C_DIS
LIN {X -0.204,Y -646.970,Z 537.322,A 0.000,B 0.000,C 90.000,E1 94.012} C_DIS
LIN {X 0.230,Y -649.976,Z 537.317,A 0.000,B 0.000,C 90.000,E1 92.980} C_DIS
LIN {X 0.240,Y -651.827,Z 537.313,A 0.000,B 0.000,C 90.000,E1 92.236} C_DIS
LIN {X 0.293,Y -653.299,Z 537.308,A 0.000,B 0.000,C 90.000,E1 91.489} C_DIS
LIN {X -0.313,Y -654.410,Z 537.304,A 0.000,B 0.000,C 90.000,E1 90.802} C_DIS
LIN {X -0.251,Y -655.140,Z 537.300,A 0.000,B 0.000,C 90.000,E1 90.057} C_DIS
LIN {X -0.183,Y -655.481,Z 537.296,A 0.000,B 0.000,C 90.000,E1 89.312} C_DIS
LIN {X 0.082,Y -655.539,Z 537.293,A 0.000,B 0.000,C 90.000,E1 88.797} C_DIS
LIN {X 0.171,Y -655.349,Z 537.289,A 0.000,B 0.000,C 90.000,E1 88.051} C_DIS
LIN {X 0.238,Y -654.841,Z 537.285,A 0.000,B 0.000,C 90.000,E1 87.306} C_DIS
LIN {X 0.326,Y -653.974,Z 537.281,A 0.000,B 0.000,C 90.000,E1 86.560} C_DIS
LIN {X 0.203,Y -652.423,Z 537.276,A 0.000,B 0.000,C 90.000,E1 85.584} C_DIS
LIN {X 0.051,Y -650.303,Z 537.270,A 0.000,B 0.000,C 90.000,E1 84.609} C_DIS
LIN {X 0.159,Y -648.506,Z 537.266,A 0.000,B 0.000,C 90.000,E1 83.856} C_DIS
LIN {X 0.181,Y -646.405,Z 537.262,A 0.000,B 0.000,C 90.000,E1 83.109} C_DIS
LIN {X -0.220,Y -644.869,Z 537.259,A 0.000,B 0.000,C 90.000,E1 82.648} C_DIS
LIN {X 0.316,Y -641.414,Z 537.254,A 0.000,B 0.000,C 90.000,E1 81.602} C_DIS
LIN {X 0.348,Y -638.527,Z 537.249,A 0.000,B 0.000,C 90.000,E1 80.849} C_DIS
LIN {X -0.277,Y -635.376,Z 537.245,A 0.000,B 0.000,C 90.000,E1 80.151} C_DIS
LIN {X -0.305,Y -631.875,Z 537.241,A 0.000,B 0.000,C 90.000,E1 79.398} C_DIS
LIN {X -0.218,Y -628.864,Z 537.237,A 0.000,B 0.000,C 90.000,E1 78.757} C_DIS
LIN {X -0.161,Y -625.727,Z 537.234,A 0.000,B 0.000,C 90.000,E1 78.117} C_DIS
LIN {X 0.207,Y -623.671,Z 537.232,A 0.000,B 0.000,C 90.000,E1 77.701} C_DIS
LIN {X -0.177,Y -621.539,Z 537.230,A 0.000,B 0.000,C 90.000,E1 77.353} C_DIS
LIN {X -0.275,Y -618.966,Z 537.227,A 0.000,B 0.000,C 90.000,E1 76.881} C_DIS
LIN {X -0.124,Y -615.928,Z 537.224,A 0.000,B 0.000,C 90.000,E1 76.353} C_DIS
LIN {X -0.088,Y -610.897,Z 537.220,A 0.000,B 0.000,C 90.000,E1 75.574} C_DIS
LIN {X 0.256,Y -608.903,Z 537.218,A 0.000,B 0.000,C 90.000,E1 75.283} C_DIS
LIN {X 0.197,Y -605.562,Z 537.216,A 0.000,B 0.000,C 90.000,E1 74.810} C_DIS
LIN {X 0.188,Y -600.358,Z 537.212,A 0.000,B 0.000,C 90.000,E1 74.157} C_DIS
LIN {X -0.050,Y -596.102,Z 537.209,A 0.000,B 0.000,C 90.000,E1 73.685} C_DIS
LIN {X 0.105,Y -589.833,Z 537.206,A 0.000,B 0.000,C 90.000,E1 73.015} C_DIS
LIN {X -0.294,Y -584.545,Z 537.203,A 0.000,B 0.000,C 90.000,E1 72.543} C_DIS
LIN {X 0.288,Y -578.906,Z 537.200,A 0.000,B 0.000,C 90.000,E1 72.000} C_DIS
LIN {X -0.151,Y -574.651,Z 537.198,A 0.000,B 0.000,C 90.000,E1 71.692} C_DIS
LIN {X 0.063,Y -568.683,Z 537.196,A 0.000,B 0.000,C 90.000,E1 71.221} C_DIS
LIN {X 0.151,Y -562.391,Z 537.193,A 0.000,B 0.000,C 90.000,E1 70.786} C_DIS
LIN {X 0.041,Y -557.542,Z 537.192,A 0.000,B 0.000,C 90.000,E1 70.496} C_DIS
LIN {X 0.129,Y -550.773,Z 537.190,A 0.000,B 0.000,C 90.000,E1 70.115} C_DIS
LIN {X -0.149,Y -543.730,Z 537.188,A 0.000,B 0.000,C 90.000,E1 69.806} C_DIS
LIN {X -0.109,Y -538.374,Z 537.187,A 0.000,B 0.000,C 90.000,E1 69.571} C_DIS
LIN {X 0.106,Y -532.956,Z 537.185,A 0.000,B 0.000,C 90.000,E1 69.337} C_DIS
LIN {X 0.194,Y -522.000,Z 537.183,A 0.000,B 0.000,C 90.000,E1 68.954} C_DIS
LIN {X 0.194,Y -514.845,Z 537.182,A 0.000,B 0.000,C 90.000,E1 68.720} C_DIS
LIN {X 0.102,Y -504.029,Z 537.180,A 0.000,B 0.000,C 90.000,E1 68.411} C_DIS
LIN {X -0.109,Y -496.587,Z 537.179,A 0.000,B 0.000,C 90.000,E1 68.230} C_DIS
LIN {X 0.034,Y -466.194,Z 537.175,A 0.000,B 0.000,C 90.000,E1 67.411} C_DIS
LIN {X 0.010,Y -466.125,Z 537.175,A 0.000,B 0.000,C 90.000,E1 67.411} C_DIS
LIN {X 0.088,Y -465.644,Z 537.173,A 0.000,B 0.000,C 90.000,E1 67.050} C_DIS
LIN {X -0.033,Y -456.637,Z 537.148,A 0.000,B 0.000,C 90.000,E1 62.615} C_DIS
LIN {X -0.034,Y -455.594,Z 537.144,A 0.000,B 0.000,C 90.000,E1 61.975} C_DIS
LIN {X 0.150,Y -452.503,Z 537.137,A 0.000,B 0.000,C 90.000,E1 60.667} C_DIS
LIN {X -0.214,Y -443.902,Z 537.114,A 0.000,B 0.000,C 90.000,E1 56.501} C_DIS
LIN {X -0.037,Y -443.434,Z 537.113,A 0.000,B 0.000,C 90.000,E1 56.294} C_DIS
LIN {X -0.075,Y -443.429,Z 537.113,A 0.000,B 0.000,C 90.000,E1 56.294} C_DIS
LIN {X -0.117,Y -445.847,Z 537.107,A 0.000,B 0.000,C 90.000,E1 55.182} C_DIS
LIN {X -0.048,Y -447.858,Z 537.101,A 0.000,B 0.000,C 90.000,E1 54.196} C_DIS
LIN {X 0.018,Y -450.478,Z 537.094,A 0.000,B 0.000,C 90.000,E1 52.889} C_DIS
LIN {X -0.148,Y -452.832,Z 537.087,A 0.000,B 0.000,C 90.000,E1 51.618} C_DIS
LIN {X -0.010,Y -454.984,Z 537.080,A 0.000,B 0.000,C 90.000,E1 50.312} C_DIS
LIN {X -0.263,Y -456.552,Z 537.074,A 0.000,B 0.000,C 90.000,E1 49.380} C_DIS
LIN {X -0.088,Y -458.856,Z 537.065,A 0.000,B 0.000,C 90.000,E1 47.757} C_DIS
LIN {X 0.089,Y -460.348,Z 537.058,A 0.000,B 0.000,C 90.000,E1 46.458} C_DIS
LIN {X 0.223,Y -461.225,Z 537.053,A 0.000,B 0.000,C 90.000,E1 45.486} C_DIS
LIN {X -0.235,Y -462.095,Z 537.046,A 0.000,B 0.000,C 90.000,E1 44.271} C_DIS
LIN {X -0.082,Y -462.599,Z 537.041,A 0.000,B 0.000,C 90.000,E1 43.299} C_DIS
LIN {X 0.099,Y -462.984,Z 537.035,A 0.000,B 0.000,C 90.000,E1 42.324} C_DIS
LIN {X -0.004,Y -463.222,Z 537.028,A 0.000,B 0.000,C 90.000,E1 41.067} C_DIS
LIN {X -0.059,Y -463.199,Z 537.021,A 0.000,B 0.000,C 90.000,E1 39.806} C_DIS
LIN {X -0.114,Y -462.992,Z 537.014,A 0.000,B 0.000,C 90.000,E1 38.543} C_DIS
LIN {X 0.190,Y -462.578,Z 537.007,A 0.000,B 0.000,C 90.000,E1 37.237} C_DIS
LIN {X -0.164,Y -462.099,Z 537.000,A 0.000,B 0.000,C 90.000,E1 36.011} C_DIS
LIN {X -0.163,Y -461.077,Z 536.988,A 0.000,B 0.000,C 90.000,E1 33.785} C_DIS
LIN {X -0.043,Y -460.475,Z 536.981,A 0.000,B 0.000,C 90.000,E1 32.498} C_DIS
LIN {X -0.201,Y -459.740,Z 536.972,A 0.000,B 0.000,C 90.000,E1 30.924} C_DIS
LIN {X -0.108,Y -458.737,Z 536.961,A 0.000,B 0.000,C 90.000,E1 28.999} C_DIS
LIN {X -0.071,Y -457.765,Z 536.950,A 0.000,B 0.000,C 90.000,E1 27.078} C_DIS
LIN {X 0.048,Y -456.670,Z 536.938,A 0.000,B 0.000,C 90.000,E1 24.823} C_DIS
LIN {X 0.071,Y -455.847,Z 536.927,A 0.000,B 0.000,C 90.000,E1 22.898} C_DIS
LIN {X 0.180,Y -455.336,Z 536.918,A 0.000,B 0.000,C 90.000,E1 21.280} C_DIS
LIN {X 0.073,Y -454.666,Z 536.904,A 0.000,B 0.000,C 90.000,E1 18.725} C_DIS
LIN {X 0.019,Y -454.330,Z 536.893,A 0.000,B 0.000,C 90.000,E1 16.804} C_DIS
LIN {X -0.085,Y -454.272,Z 536.879,A 0.000,B 0.000,C 90.000,E1 14.245} C_DIS
LIN {X 0.102,Y -454.787,Z 536.861,A 0.000,B 0.000,C 90.000,E1 11.007} C_DIS
LIN {X 0.190,Y -455.794,Z 536.845,A 0.000,B 0.000,C 90.000,E1 8.106} C_DIS
LIN {X -0.023,Y -457.066,Z 536.831,A 0.000,B 0.000,C 90.000,E1 5.568} C_DIS
LIN {X -0.004,Y -458.548,Z 536.819,A 0.000,B 0.000,C 90.000,E1 3.326} C_DIS
LIN {X 0.223,Y -460.591,Z 536.804,A 0.000,B 0.000,C 90.000,E1 0.745} C_DIS
LIN {X 0.059,Y -463.681,Z 536.788,A 0.000,B 0.000,C 90.000,E1 357.879} C_DIS
LIN {X -0.010,Y -466.828,Z 536.774,A 0.000,B 0.000,C 90.000,E1 355.355} C_DIS
LIN {X -0.175,Y -468.855,Z 536.766,A 0.000,B 0.000,C 90.000,E1 353.799} C_DIS
LIN {X -0.054,Y -470.520,Z 536.758,A 0.000,B 0.000,C 90.000,E1 352.527} C_DIS
LIN {X -0.152,Y -472.671,Z 536.750,A 0.000,B 0.000,C 90.000,E1 350.971} C_DIS
LIN {X -0.233,Y -475.322,Z 536.739,A 0.000,B 0.000,C 90.000,E1 349.106} C_DIS
LIN {X -0.178,Y -480.317,Z 536.722,A 0.000,B 0.000,C 90.000,E1 345.992} C_DIS
LIN {X 0.121,Y -484.302,Z 536.710,A 0.000,B 0.000,C 90.000,E1 343.795} C_DIS
LIN {X 0.059,Y -489.072,Z 536.696,A 0.000,B 0.000,C 90.000,E1 341.348} C_DIS
LIN {X 0.063,Y -492.689,Z 536.686,A 0.000,B 0.000,C 90.000,E1 339.518} C_DIS
LIN {X -0.179,Y -495.657,Z 536.678,A 0.000,B 0.000,C 90.000,E1 338.028} C_DIS
LIN {X 0.039,Y -498.032,Z 536.671,A 0.000,B 0.000,C 90.000,E1 336.794} C_DIS
LIN {X -0.174,Y -500.374,Z 536.664,A 0.000,B 0.000,C 90.000,E1 335.613} C_DIS
LIN {X 0.144,Y -503.155,Z 536.656,A 0.000,B 0.000,C 90.000,E1 334.076} C_DIS
LIN {X 0.152,Y -506.484,Z 536.646,A 0.000,B 0.000,C 90.000,E1 332.281} C_DIS
LIN {X 0.103,Y -510.197,Z 536.635,A 0.000,B 0.000,C 90.000,E1 330.205} C_DIS
LIN {X -0.136,Y -513.436,Z 536.625,A 0.000,B 0.000,C 90.000,E1 328.456} C_DIS
LIN {X 0.053,Y -516.143,Z 536.617,A 0.000,B 0.000,C 90.000,E1 326.962} C_DIS
LIN {X -0.141,Y -518.910,Z 536.608,A 0.000,B 0.000,C 90.000,E1 325.515} C_DIS
LIN {X 0.011,Y -521.629,Z 536.600,A 0.000,B 0.000,C 90.000,E1 324.036} C_DIS
LIN {X 0.095,Y -525.973,Z 536.587,A 0.000,B 0.000,C 90.000,E1 321.698} C_DIS
LIN {X -0.167,Y -529.279,Z 536.578,A 0.000,B 0.000,C 90.000,E1 319.989} C_DIS
LIN {X -0.085,Y -534.035,Z 536.565,A 0.000,B 0.000,C 90.000,E1 317.676} C_DIS
LIN {X 0.143,Y -538.404,Z 536.554,A 0.000,B 0.000,C 90.000,E1 315.648} C_DIS
LIN {X -0.285,Y -545.096,Z 536.538,A 0.000,B 0.000,C 90.000,E1 312.852} C_DIS
LIN {X -0.181,Y -549.237,Z 536.529,A 0.000,B 0.000,C 90.000,E1 311.148} C_DIS
LIN {X -0.099,Y -551.150,Z 536.524,A 0.000,B 0.000,C 90.000,E1 310.297} C_DIS
LIN {X -0.293,Y -553.546,Z 536.518,A 0.000,B 0.000,C 90.000,E1 309.197} C_DIS
LIN {X -0.220,Y -557.886,Z 536.507,A 0.000,B 0.000,C 90.000,E1 307.237} C_DIS
LIN {X 0.073,Y -558.992,Z 536.504,A 0.000,B 0.000,C 90.000,E1 306.790} C_DIS
LIN {X -0.058,Y -560.323,Z 536.503,A 0.000,B 0.000,C 90.000,E1 306.503} C_DIS
LIN {X -0.192,Y -561.388,Z 536.501,A 0.000,B 0.000,C 90.000,E1 306.171} C_DIS
LIN {X 0.011,Y -563.559,Z 536.499,A 0.000,B 0.000,C 90.000,E1 305.804} C_DIS
LIN {X -0.103,Y -564.198,Z 536.498,A 0.000,B 0.000,C 90.000,E1 305.678} C_DIS
LIN {X -0.045,Y -569.169,Z 536.495,A 0.000,B 0.000,C 90.000,E1 305.025} C_DIS
LIN {X 0.078,Y -573.653,Z 536.492,A 0.000,B 0.000,C 90.000,E1 304.485} C_DIS
LIN {X 0.001,Y -585.876,Z 536.484,A 0.000,B 0.000,C 90.000,E1 303.166} C_DIS
LIN {X 0.349,Y -597.889,Z 536.477,A 0.000,B 0.000,C 90.000,E1 301.799} C_DIS
LIN {X -0.143,Y -606.038,Z 536.472,A 0.000,B 0.000,C 90.000,E1 300.924} C_DIS
LIN {X -0.237,Y -609.313,Z 536.470,A 0.000,B 0.000,C 90.000,E1 300.541} C_DIS
LIN {X -0.073,Y -616.561,Z 536.465,A 0.000,B 0.000,C 90.000,E1 299.617} C_DIS
LIN {X 0.176,Y -622.438,Z 536.460,A 0.000,B 0.000,C 90.000,E1 298.693} C_DIS
LIN {X 0.175,Y -623.977,Z 536.458,A 0.000,B 0.000,C 90.000,E1 298.437} C_DIS
LIN {X -0.058,Y -627.568,Z 536.454,A 0.000,B 0.000,C 90.000,E1 297.692} C_DIS
LIN {X -0.005,Y -629.927,Z 536.450,A 0.000,B 0.000,C 90.000,E1 296.924} C_DIS
LIN {X 0.073,Y -630.638,Z 536.445,A 0.000,B 0.000,C 90.000,E1 296.155} C_DIS
LIN {X -0.143,Y -630.343,Z 536.443,A 0.000,B 0.000,C 90.000,E1 295.668} C_DIS
LIN {X -0.113,Y -629.936,Z 536.441,A 0.000,B 0.000,C 90.000,E1 295.412} C_DIS
LIN {X -0.057,Y -628.427,Z 536.438,A 0.000,B 0.000,C 90.000,E1 294.899} C_DIS
LIN {X -0.015,Y -625.266,Z 536.436,A 0.000,B 0.000,C 90.000,E1 294.387} C_DIS
LIN {X -0.009,Y -624.351,Z 536.435,A 0.000,B 0.000,C 90.000,E1 294.259} C_DIS
LIN {X -0.003,Y -622.692,Z 536.434,A 0.000,B 0.000,C 90.000,E1 294.131} C_DIS
LIN {X -0.252,Y -619.261,Z 536.432,A 0.000,B 0.000,C 90.000,E1 293.823} C_DIS
LIN {X -0.185,Y -617.673,Z 536.432,A 0.000,B 0.000,C 90.000,E1 293.695} C_DIS
LIN {X 0.295,Y -610.879,Z 536.429,A 0.000,B 0.000,C 90.000,E1 293.259} C_DIS
LIN {X 0.040,Y -605.015,Z 536.428,A 0.000,B 0.000,C 90.000,E1 293.025} C_DIS
LIN {X 0.065,Y -603.817,Z 536.428,A 0.000,B 0.000,C 90.000,E1 292.950} C_DIS
LIN {X 0.140,Y -601.850,Z 536.427,A 0.000,B 0.000,C 90.000,E1 292.845} C_DIS
LIN {X -0.185,Y -594.622,Z 536.425,A 0.000,B 0.000,C 90.000,E1 292.589} C_DIS
LIN {X -0.289,Y -590.658,Z 536.425,A 0.000,B 0.000,C 90.000,E1 292.461} C_DIS
LIN {X -0.229,Y -583.451,Z 536.423,A 0.000,B 0.000,C 90.000,E1 292.153} C_DIS
LIN {X 0.006,Y -578.832,Z 536.422,A 0.000,B 0.000,C 90.000,E1 291.897} C_DIS
LIN {X -0.142,Y -574.999,Z 536.420,A 0.000,B 0.000,C 90.000,E1 291.642} C_DIS
LIN {X -0.094,Y -573.781,Z 536.419,A 0.000,B 0.000,C 90.000,E1 291.461} C_DIS
LIN {X 0.212,Y -573.349,Z 536.418,A 0.000,B 0.000,C 90.000,E1 291.227} C_DIS
LIN {X -0.036,Y -573.059,Z 536.416,A 0.000,B 0.000,C 90.000,E1 290.791} C_DIS
LIN {X 0.120,Y -573.282,Z 536.406,A 0.000,B 0.000,C 90.000,E1 289.141} C_DIS
LIN {X 0.100,Y -573.253,Z 536.400,A 0.000,B 0.000,C 90.000,E1 288.055} C_DIS
LIN {X -0.091,Y -573.104,Z 536.394,A 0.000,B 0.000,C 90.000,E1 286.985} C_DIS
LIN {X -0.118,Y -572.832,Z 536.388,A 0.000,B 0.000,C 90.000,E1 285.898} C_DIS
LIN {X 0.070,Y -572.098,Z 536.379,A 0.000,B 0.000,C 90.000,E1 284.245} C_DIS
LIN {X 0.245,Y -571.358,Z 536.370,A 0.000,B 0.000,C 90.000,E1 282.591} C_DIS
LIN {X 0.083,Y -570.722,Z 536.363,A 0.000,B 0.000,C 90.000,E1 281.243} C_DIS
LIN {X -0.200,Y -570.007,Z 536.355,A 0.000,B 0.000,C 90.000,E1 279.905} C_DIS
LIN {X 0.250,Y -569.242,Z 536.346,A 0.000,B 0.000,C 90.000,E1 278.219} C_DIS
LIN {X 0.133,Y -568.445,Z 536.335,A 0.000,B 0.000,C 90.000,E1 276.315} C_DIS
LIN {X 0.234,Y -567.998,Z 536.328,A 0.000,B 0.000,C 90.000,E1 274.935} C_DIS
LIN {X -0.239,Y -567.373,Z 536.320,A 0.000,B 0.000,C 90.000,E1 273.612} C_DIS
LIN {X -0.077,Y -566.372,Z 536.311,A 0.000,B 0.000,C 90.000,E1 271.949} C_DIS
LIN {X -0.165,Y -565.709,Z 536.305,A 0.000,B 0.000,C 90.000,E1 270.859} C_DIS
LIN {X -0.274,Y -564.917,Z 536.299,A 0.000,B 0.000,C 90.000,E1 269.771} C_DIS
LIN {X -0.059,Y -563.465,Z 536.288,A 0.000,B 0.000,C 90.000,E1 267.822} C_DIS
LIN {X 0.242,Y -561.861,Z 536.276,A 0.000,B 0.000,C 90.000,E1 265.584} C_DIS
LIN {X 0.138,Y -560.959,Z 536.270,A 0.000,B 0.000,C 90.000,E1 264.489} C_DIS
LIN {X 0.100,Y -559.743,Z 536.262,A 0.000,B 0.000,C 90.000,E1 263.109} C_DIS
LIN {X 0.096,Y -558.500,Z 536.254,A 0.000,B 0.000,C 90.000,E1 261.724} C_DIS
LIN {X -0.037,Y -557.706,Z 536.250,A 0.000,B 0.000,C 90.000,E1 260.905} C_DIS
LIN {X 0.012,Y -555.989,Z 536.242,A 0.000,B 0.000,C 90.000,E1 259.511} C_DIS
LIN {X 0.018,Y -554.320,Z 536.234,A 0.000,B 0.000,C 90.000,E1 258.117} C_DIS
LIN {X 0.221,Y -552.475,Z 536.226,A 0.000,B 0.000,C 90.000,E1 256.700} C_DIS
LIN {X -0.136,Y -550.438,Z 536.219,A 0.000,B 0.000,C 90.000,E1 255.338} C_DIS
LIN {X -0.098,Y -548.668,Z 536.212,A 0.000,B 0.000,C 90.000,E1 254.212} C_DIS
LIN {X -0.094,Y -546.781,Z 536.206,A 0.000,B 0.000,C 90.000,E1 253.087} C_DIS
LIN {X 0.036,Y -544.737,Z 536.200,A 0.000,B 0.000,C 90.000,E1 251.945} C_DIS
LIN {X -0.145,Y -541.985,Z 536.192,A 0.000,B 0.000,C 90.000,E1 250.550} C_DIS
LIN {X 0.092,Y -539.642,Z 536.186,A 0.000,B 0.000,C 90.000,E1 249.390} C_DIS
LIN {X 0.009,Y -536.577,Z 536.178,A 0.000,B 0.000,C 90.000,E1 247.975} C_DIS
LIN {X -0.129,Y -533.986,Z 536.171,A 0.000,B 0.000,C 90.000,E1 246.847} C_DIS
LIN {X 0.187,Y -531.172,Z 536.165,A 0.000,B 0.000,C 90.000,E1 245.665} C_DIS
LIN {X -0.211,Y -528.991,Z 536.160,A 0.000,B 0.000,C 90.000,E1 244.845} C_DIS
LIN {X 0.243,Y -525.945,Z 536.154,A 0.000,B 0.000,C 90.000,E1 243.640} C_DIS
LIN {X -0.140,Y -521.948,Z 536.146,A 0.000,B 0.000,C 90.000,E1 242.231} C_DIS
LIN {X 0.102,Y -517.912,Z 536.138,A 0.000,B 0.000,C 90.000,E1 240.745} C_DIS
LIN {X -0.032,Y -514.626,Z 536.131,A 0.000,B 0.000,C 90.000,E1 239.587} C_DIS
LIN {X -0.025,Y -511.183,Z 536.125,A 0.000,B 0.000,C 90.000,E1 238.408} C_DIS
LIN {X -0.015,Y -505.842,Z 536.115,A 0.000,B 0.000,C 90.000,E1 236.628} C_DIS
LIN {X 0.162,Y -500.462,Z 536.105,A 0.000,B 0.000,C 90.000,E1 234.815} C_DIS
LIN {X -0.053,Y -496.189,Z 536.096,A 0.000,B 0.000,C 90.000,E1 233.336} C_DIS
LIN {X -0.201,Y -491.130,Z 536.086,A 0.000,B 0.000,C 90.000,E1 231.537} C_DIS
LIN {X -0.023,Y -485.344,Z 536.074,A 0.000,B 0.000,C 90.000,E1 229.380} C_DIS
LIN {X -0.174,Y -480.522,Z 536.064,A 0.000,B 0.000,C 90.000,E1 227.553} C_DIS
LIN {X -0.012,Y -475.110,Z 536.052,A 0.000,B 0.000,C 90.000,E1 225.364} C_DIS
LIN {X 0.059,Y -471.991,Z 536.045,A 0.000,B 0.000,C 90.000,E1 224.109} C_DIS
LIN {X -0.070,Y -467.593,Z 536.035,A 0.000,B 0.000,C 90.000,E1 222.243} C_DIS
LIN {X 0.052,Y -463.199,Z 536.024,A 0.000,B 0.000,C 90.000,E1 220.334} C_DIS
LIN {X -0.231,Y -458.932,Z 536.014,A 0.000,B 0.000,C 90.000,E1 218.463} C_DIS
LIN {X 0.099,Y -454.780,Z 536.003,A 0.000,B 0.000,C 90.000,E1 216.503} C_DIS
LIN {X 0.208,Y -449.400,Z 535.989,A 0.000,B 0.000,C 90.000,E1 213.913} C_DIS
LIN {X -0.098,Y -445.527,Z 535.978,A 0.000,B 0.000,C 90.000,E1 212.005} C_DIS
LIN {X 0.154,Y -443.040,Z 535.971,A 0.000,B 0.000,C 90.000,E1 210.669} C_DIS
LIN {X -0.111,Y -438.835,Z 535.958,A 0.000,B 0.000,C 90.000,E1 208.409} C_DIS
LIN {X -0.134,Y -434.862,Z 535.945,A 0.000,B 0.000,C 90.000,E1 206.104} C_DIS
LIN {X -0.055,Y -431.040,Z 535.932,A 0.000,B 0.000,C 90.000,E1 203.770} C_DIS
LIN {X 0.139,Y -427.442,Z 535.919,A 0.000,B 0.000,C 90.000,E1 201.408} C_DIS
LIN {X -0.103,Y -423.270,Z 535.902,A 0.000,B 0.000,C 90.000,E1 198.417} C_DIS
LIN {X -0.073,Y -420.699,Z 535.891,A 0.000,B 0.000,C 90.000,E1 196.386} C_DIS
LIN {X 0.142,Y -418.697,Z 535.882,A 0.000,B 0.000,C 90.000,E1 194.662} C_DIS
LIN {X 0.158,Y -417.024,Z 535.874,A 0.000,B 0.000,C 90.000,E1 193.300} C_DIS
LIN {X 0.184,Y -414.899,Z 535.865,A 0.000,B 0.000,C 90.000,E1 191.591} C_DIS
LIN {X 0.001,Y -412.942,Z 535.855,A 0.000,B 0.000,C 90.000,E1 189.905} C_DIS
LIN {X 0.220,Y -410.676,Z 535.844,A 0.000,B 0.000,C 90.000,E1 187.814} C_DIS
LIN {X -0.119,Y -408.175,Z 535.830,A 0.000,B 0.000,C 90.000,E1 185.448} C_DIS
LIN {X 0.208,Y -406.016,Z 535.817,A 0.000,B 0.000,C 90.000,E1 182.980} C_DIS
LIN {X -0.055,Y -403.416,Z 535.797,A 0.000,B 0.000,C 90.000,E1 179.542} C_DIS
LIN {X 0.110,Y -402.178,Z 535.784,A 0.000,B 0.000,C 90.000,E1 177.078} C_DIS
LIN {X -0.136,Y -401.274,Z 535.768,A 0.000,B 0.000,C 90.000,E1 174.318} C_DIS
LIN {X 0.079,Y -400.868,Z 535.753,A 0.000,B 0.000,C 90.000,E1 171.489} C_DIS
LIN {X 0.030,Y -400.881,Z 535.743,A 0.000,B 0.000,C 90.000,E1 169.746} C_DIS
LIN {X 0.044,Y -401.103,Z 535.731,A 0.000,B 0.000,C 90.000,E1 167.645} C_DIS
LIN {X -0.081,Y -401.714,Z 535.716,A 0.000,B 0.000,C 90.000,E1 164.866} C_DIS
LIN {X -0.149,Y -402.453,Z 535.704,A 0.000,B 0.000,C 90.000,E1 162.779} C_DIS
LIN {X -0.185,Y -403.232,Z 535.695,A 0.000,B 0.000,C 90.000,E1 161.040} C_DIS
LIN {X -0.024,Y -404.734,Z 535.679,A 0.000,B 0.000,C 90.000,E1 158.230} C_DIS
LIN {X 0.026,Y -405.775,Z 535.669,A 0.000,B 0.000,C 90.000,E1 156.485} C_DIS
LIN {X -0.006,Y -407.168,Z 535.658,A 0.000,B 0.000,C 90.000,E1 154.409} C_DIS
LIN {X 0.078,Y -408.377,Z 535.648,A 0.000,B 0.000,C 90.000,E1 152.666} C_DIS
LIN {X 0.188,Y -409.529,Z 535.639,A 0.000,B 0.000,C 90.000,E1 150.923} C_DIS
LIN {X -0.122,Y -410.361,Z 535.631,A 0.000,B 0.000,C 90.000,E1 149.587} C_DIS
LIN {X -0.139,Y -411.207,Z 535.621,A 0.000,B 0.000,C 90.000,E1 147.867} C_DIS
LIN {X -0.050,Y -411.988,Z 535.612,A 0.000,B 0.000,C 90.000,E1 146.135} C_DIS
LIN {X 0.058,Y -412.585,Z 535.602,A 0.000,B 0.000,C 90.000,E1 144.402} C_DIS
LIN {X 0.082,Y -413.099,Z 535.593,A 0.000,B 0.000,C 90.000,E1 142.683} C_DIS
LIN {X 0.111,Y -413.460,Z 535.583,A 0.000,B 0.000,C 90.000,E1 140.964} C_DIS
LIN {X 0.074,Y -413.744,Z 535.574,A 0.000,B 0.000,C 90.000,E1 139.256} C_DIS
LIN {X -0.134,Y -413.886,Z 535.562,A 0.000,B 0.000,C 90.000,E1 137.229} C_DIS
LIN {X 0.084,Y -413.959,Z 535.553,A 0.000,B 0.000,C 90.000,E1 135.486} C_DIS
LIN {X 0.139,Y -414.032,Z 535.545,A 0.000,B 0.000,C 90.000,E1 134.109} C_DIS
LIN {X -0.092,Y -413.981,Z 535.538,A 0.000,B 0.000,C 90.000,E1 132.771} C_DIS
LIN {X -0.019,Y -413.833,Z 535.530,A 0.000,B 0.000,C 90.000,E1 131.391} C_DIS
LIN {X 0.050,Y -413.482,Z 535.522,A 0.000,B 0.000,C 90.000,E1 130.011} C_DIS
LIN {X -0.159,Y -412.830,Z 535.515,A 0.000,B 0.000,C 90.000,E1 128.669} C_DIS
LIN {X -0.004,Y -411.969,Z 535.506,A 0.000,B 0.000,C 90.000,E1 127.156} C_DIS
LIN {X -0.043,Y -411.978,Z 535.506,A 0.000,B 0.000,C 90.000,E1 127.156} C_DIS
LIN {X 0.123,Y -415.720,Z 535.500,A 0.000,B 0.000,C 90.000,E1 125.884} C_DIS
LIN {X 0.230,Y -425.158,Z 535.479,A 0.000,B 0.000,C 90.000,E1 122.133} C_DIS
LIN {X 0.165,Y -430.154,Z 535.469,A 0.000,B 0.000,C 90.000,E1 120.463} C_DIS
LIN {X 0.163,Y -431.085,Z 535.468,A 0.000,B 0.000,C 90.000,E1 120.129} C_DIS
LIN {X 0.111,Y -440.177,Z 535.447,A 0.000,B 0.000,C 90.000,E1 116.488} C_DIS
LIN {X 0.117,Y -444.941,Z 535.438,A 0.000,B 0.000,C 90.000,E1 114.847} C_DIS
LIN {X -0.041,Y -448.409,Z 535.429,A 0.000,B 0.000,C 90.000,E1 113.259} C_DIS
LIN {X -0.081,Y -448.450,Z 535.429,A 0.000,B 0.000,C 90.000,E1 113.259} C_DIS
LIN {X 0.189,Y -478.820,Z 535.423,A 0.000,B 0.000,C 90.000,E1 112.025} C_DIS
LIN {X -0.037,Y -487.511,Z 535.421,A 0.000,B 0.000,C 90.000,E1 111.716} C_DIS
LIN {X 0.223,Y -504.646,Z 535.417,A 0.000,B 0.000,C 90.000,E1 110.972} C_DIS
LIN {X -0.265,Y -518.283,Z 535.413,A 0.000,B 0.000,C 90.000,E1 110.429} C_DIS
LIN {X -0.147,Y -524.794,Z 535.412,A 0.000,B 0.000,C 90.000,E1 110.120} C_DIS
LIN {X 0.222,Y -531.525,Z 535.410,A 0.000,B 0.000,C 90.000,E1 109.758} C_DIS
LIN {X 0.032,Y -538.057,Z 535.408,A 0.000,B 0.000,C 90.000,E1 109.450} C_DIS
LIN {X -0.152,Y -546.041,Z 535.406,A 0.000,B 0.000,C 90.000,E1 109.033} C_DIS
LIN {X 0.139,Y -550.680,Z 535.404,A 0.000,B 0.000,C 90.000,E1 108.725} C_DIS
LIN {X -0.038,Y -553.848,Z 535.403,A 0.000,B 0.000,C 90.000,E1 108.544} C_DIS
LIN {X 0.047,Y -559.678,Z 535.401,A 0.000,B 0.000,C 90.000,E1 108.127} C_DIS
LIN {X 0.335,Y -564.849,Z 535.399,A 0.000,B 0.000,C 90.000,E1 107.692} C_DIS
LIN {X 0.296,Y -567.147,Z 535.398,A 0.000,B 0.000,C 90.000,E1 107.511} C_DIS
LIN {X 0.220,Y -572.483,Z 535.395,A 0.000,B 0.000,C 90.000,E1 107.040} C_DIS
LIN {X -0.248,Y -577.294,Z 535.392,A 0.000,B 0.000,C 90.000,E1 106.622} C_DIS
LIN {X 0.073,Y -580.758,Z 535.390,A 0.000,B 0.000,C 90.000,E1 106.205} C_DIS
LIN {X -0.020,Y -582.094,Z 535.389,A 0.000,B 0.000,C 90.000,E1 106.079} C_DIS
LIN {X -0.210,Y -588.774,Z 535.385,A 0.000,B 0.000,C 90.000,E1 105.300} C_DIS
LIN {X -0.079,Y -592.723,Z 535.382,A 0.000,B 0.000,C 90.000,E1 104.773} C_DIS
LIN {X 0.172,Y -598.277,Z 535.378,A 0.000,B 0.000,C 90.000,E1 103.953} C_DIS
LIN {X 0.042,Y -603.545,Z 535.373,A 0.000,B 0.000,C 90.000,E1 103.175} C_DIS
LIN {X -0.113,Y -607.772,Z 535.370,A 0.000,B 0.000,C 90.000,E1 102.535} C_DIS
LIN {X -0.104,Y -611.820,Z 535.366,A 0.000,B 0.000,C 90.000,E1 101.883} C_DIS
LIN {X -0.188,Y -615.620,Z 535.362,A 0.000,B 0.000,C 90.000,E1 101.243} C_DIS
LIN {X 0.197,Y -619.781,Z 535.358,A 0.000,B 0.000,C 90.000,E1 100.433} C_DIS
LIN {X 0.212,Y -622.966,Z 535.355,A 0.000,B 0.000,C 90.000,E1 99.792} C_DIS
LIN {X -0.151,Y -627.766,Z 535.349,A 0.000,B 0.000,C 90.000,E1 98.803} C_DIS
LIN {X 0.166,Y -632.254,Z 535.343,A 0.000,B 0.000,C 90.000,E1 97.757} C_DIS
LIN {X -0.174,Y -636.743,Z 535.338,A 0.000,B 0.000,C 90.000,E1 96.777} C_DIS
LIN {X 0.179,Y -641.043,Z 535.332,A 0.000,B 0.000,C 90.000,E1 95.739} C_DIS
LIN {X -0.053,Y -644.872,Z 535.326,A 0.000,B 0.000,C 90.000,E1 94.759} C_DIS
LIN {X -0.064,Y -647.452,Z 535.322,A 0.000,B 0.000,C 90.000,E1 94.012} C_DIS
LIN {X -0.271,Y -650.488,Z 535.317,A 0.000,B 0.000,C 90.000,E1 93.037} C_DIS
LIN {X -0.259,Y -652.355,Z 535.313,A 0.000,B 0.000,C 90.000,E1 92.293} C_DIS
LIN {X -0.201,Y -653.881,Z 535.309,A 0.000,B 0.000,C 90.000,E1 91.547} C_DIS
LIN {X 0.051,Y -654.672,Z 535.306,A 0.000,B 0.000,C 90.000,E1 91.031} C_DIS
LIN {X 0.114,Y -655.506,Z 535.302,A 0.000,B 0.000,C 90.000,E1 90.286} C_DIS
LIN {X 0.187,Y -656.011,Z 535.298,A 0.000,B 0.000,C 90.000,E1 89.542} C_DIS
LIN {X 0.263,Y -656.103,Z 535.294,A 0.000,B 0.000,C 90.000,E1 88.797} C_DIS
LIN {X -0.298,Y -655.886,Z 535.289,A 0.000,B 0.000,C 90.000,E1 88.108} C_DIS
LIN {X -0.226,Y -655.385,Z 535.285,A 0.000,B 0.000,C 90.000,E1 87.364} C_DIS
LIN {X -0.131,Y -654.494,Z 535.281,A 0.000,B 0.000,C 90.000,E1 86.617} C_DIS
LIN {X 0.118,Y -653.736,Z 535.278,A 0.000,B 0.000,C 90.000,E1 86.102} C_DIS
LIN {X 0.195,Y -652.340,Z 535.274,A 0.000,B 0.000,C 90.000,E1 85.355} C_DIS
LIN {X 0.258,Y -650.677,Z 535.270,A 0.000,B 0.000,C 90.000,E1 84.609} C_DIS
LIN {X -0.276,Y -648.835,Z 535.266,A 0.000,B 0.000,C 90.000,E1 83.913} C_DIS
LIN {X -0.248,Y -646.614,Z 535.262,A 0.000,B 0.000,C 90.000,E1 83.166} C_DIS
LIN {X -0.006,Y -645.069,Z 535.259,A 0.000,B 0.000,C 90.000,E1 82.648} C_DIS
LIN {X 0.224,Y -643.335,Z 535.256,A 0.000,B 0.000,C 90.000,E1 82.129} C_DIS
LIN {X 0.270,Y -640.517,Z 535.252,A 0.000,B 0.000,C 90.000,E1 81.376} C_DIS
LIN {X -0.068,Y -638.584,Z 535.250,A 0.000,B 0.000,C 90.000,E1 80.905} C_DIS
LIN {X -0.062,Y -635.362,Z 535.245,A 0.000,B 0.000,C 90.000,E1 80.151} C_DIS
LIN {X 0.092,Y -633.053,Z 535.242,A 0.000,B 0.000,C 90.000,E1 79.634} C_DIS
LIN {X -0.042,Y -628.104,Z 535.237,A 0.000,B 0.000,C 90.000,E1 78.634} C_DIS
LIN {X -0.198,Y -623.457,Z 535.232,A 0.000,B 0.000,C 90.000,E1 77.757} C_DIS
LIN {X 0.150,Y -617.559,Z 535.226,A 0.000,B 0.000,C 90.000,E1 76.700} C_DIS
LIN {X -0.263,Y -615.204,Z 535.224,A 0.000,B 0.000,C 90.000,E1 76.353} C_DIS
LIN {X -0.185,Y -610.907,Z 535.221,A 0.000,B 0.000,C 90.000,E1 75.700} C_DIS
LIN {X -0.193,Y -605.075,Z 535.216,A 0.000,B 0.000,C 90.000,E1 74.921} C_DIS
LIN {X -0.142,Y -600.790,Z 535.213,A 0.000,B 0.000,C 90.000,E1 74.393} C_DIS
LIN {X 0.131,Y -595.250,Z 535.210,A 0.000,B 0.000,C 90.000,E1 73.740} C_DIS
LIN {X -0.173,Y -589.080,Z 535.206,A 0.000,B 0.000,C 90.000,E1 73.142} C_DIS
LIN {X 0.193,Y -585.048,Z 535.204,A 0.000,B 0.000,C 90.000,E1 72.725} C_DIS
LIN {X -0.285,Y -579.635,Z 535.202,A 0.000,B 0.000,C 90.000,E1 72.308} C_DIS
LIN {X 0.244,Y -574.210,Z 535.199,A 0.000,B 0.000,C 90.000,E1 71.819} C_DIS
LIN {X 0.077,Y -568.373,Z 535.197,A 0.000,B 0.000,C 90.000,E1 71.402} C_DIS
LIN {X 0.144,Y -562.178,Z 535.195,A 0.000,B 0.000,C 90.000,E1 70.986} C_DIS
LIN {X 0.203,Y -557.239,Z 535.193,A 0.000,B 0.000,C 90.000,E1 70.678} C_DIS
LIN {X -0.294,Y -550.517,Z 535.191,A 0.000,B 0.000,C 90.000,E1 70.369} C_DIS
LIN {X 0.270,Y -545.307,Z 535.189,A 0.000,B 0.000,C 90.000,E1 70.061} C_DIS
LIN {X 0.272,Y -538.081,Z 535.188,A 0.000,B 0.000,C 90.000,E1 69.752} C_DIS
LIN {X 0.050,Y -532.711,Z 535.187,A 0.000,B 0.000,C 90.000,E1 69.571} C_DIS
LIN {X 0.088,Y -523.473,Z 535.185,A 0.000,B 0.000,C 90.000,E1 69.263} C_DIS
LIN {X 0.129,Y -514.578,Z 535.183,A 0.000,B 0.000,C 90.000,E1 68.975} C_DIS
LIN {X 0.058,Y -505.251,Z 535.182,A 0.000,B 0.000,C 90.000,E1 68.720} C_DIS
LIN {X 0.155,Y -496.130,Z 535.180,A 0.000,B 0.000,C 90.000,E1 68.465} C_DIS
LIN {X 0.130,Y -476.457,Z 535.178,A 0.000,B 0.000,C 90.000,E1 67.975} C_DIS
LIN {X 0.137,Y -466.685,Z 535.176,A 0.000,B 0.000,C 90.000,E1 67.720} C_DIS
LIN {X 0.091,Y -466.570,Z 535.176,A 0.000,B 0.000,C 90.000,E1 67.720} C_DIS
LIN {X -0.208,Y -465.670,Z 535.173,A 0.000,B 0.000,C 90.000,E1 67.102} C_DIS
LIN {X 0.205,Y -456.134,Z 535.146,A 0.000,B 0.000,C 90.000,E1 62.281} C_DIS
LIN {X 0.098,Y -455.620,Z 535.144,A 0.000,B 0.000,C 90.000,E1 61.975} C_DIS
LIN {X 0.085,Y -454.106,Z 535.141,A 0.000,B 0.000,C 90.000,E1 61.335} C_DIS
LIN {X 0.165,Y -445.093,Z 535.117,A 0.000,B 0.000,C 90.000,E1 57.120} C_DIS
LIN {X 0.096,Y -443.812,Z 535.114,A 0.000,B 0.000,C 90.000,E1 56.421} C_DIS
LIN {X 0.057,Y -443.812,Z 535.114,A 0.000,B 0.000,C 90.000,E1 56.421} C_DIS
LIN {X 0.021,Y -446.571,Z 535.107,A 0.000,B 0.000,C 90.000,E1 55.182} C_DIS
LIN {X 0.099,Y -448.596,Z 535.101,A 0.000,B 0.000,C 90.000,E1 54.196} C_DIS
LIN {X -0.094,Y -451.295,Z 535.094,A 0.000,B 0.000,C 90.000,E1 52.924} C_DIS
LIN {X 0.024,Y -453.657,Z 535.087,A 0.000,B 0.000,C 90.000,E1 51.618} C_DIS
LIN {X -0.173,Y -455.868,Z 535.080,A 0.000,B 0.000,C 90.000,E1 50.356} C_DIS
LIN {X -0.065,Y -457.407,Z 535.074,A 0.000,B 0.000,C 90.000,E1 49.380} C_DIS
LIN {X 0.128,Y -459.726,Z 535.065,A 0.000,B 0.000,C 90.000,E1 47.757} C_DIS
LIN {X -0.061,Y -460.873,Z 535.060,A 0.000,B 0.000,C 90.000,E1 46.824} C_DIS
LIN {X -0.240,Y -461.816,Z 535.055,A 0.000,B 0.000,C 90.000,E1 45.891} C_DIS
LIN {X -0.036,Y -462.718,Z 535.048,A 0.000,B 0.000,C 90.000,E1 44.595} C_DIS
LIN {X 0.180,Y -463.385,Z 535.041,A 0.000,B 0.000,C 90.000,E1 43.299} C_DIS
LIN {X 0.028,Y -463.784,Z 535.035,A 0.000,B 0.000,C 90.000,E1 42.366} C_DIS
LIN {X 0.280,Y -463.971,Z 535.028,A 0.000,B 0.000,C 90.000,E1 41.067} C_DIS
LIN {X -0.120,Y -463.906,Z 535.021,A 0.000,B 0.000,C 90.000,E1 39.850} C_DIS
LIN {X 0.192,Y -463.696,Z 535.014,A 0.000,B 0.000,C 90.000,E1 38.543} C_DIS
LIN {X -0.143,Y -463.290,Z 535.007,A 0.000,B 0.000,C 90.000,E1 37.317} C_DIS
LIN {X 0.163,Y -462.779,Z 535.000,A 0.000,B 0.000,C 90.000,E1 36.011} C_DIS
LIN {X 0.054,Y -461.904,Z 534.990,A 0.000,B 0.000,C 90.000,E1 34.119} C_DIS
LIN {X -0.077,Y -461.130,Z 534.981,A 0.000,B 0.000,C 90.000,E1 32.546} C_DIS
LIN {X 0.166,Y -460.364,Z 534.972,A 0.000,B 0.000,C 90.000,E1 30.924} C_DIS
LIN {X 0.051,Y -459.331,Z 534.961,A 0.000,B 0.000,C 90.000,E1 29.027} C_DIS
LIN {X -0.085,Y -458.313,Z 534.951,A 0.000,B 0.000,C 90.000,E1 27.129} C_DIS
LIN {X -0.152,Y -457.161,Z 534.938,A 0.000,B 0.000,C 90.000,E1 24.899} C_DIS
LIN {X 0.077,Y -456.582,Z 534.931,A 0.000,B 0.000,C 90.000,E1 23.590} C_DIS
LIN {X 0.111,Y -455.867,Z 534.920,A 0.000,B 0.000,C 90.000,E1 21.663} C_DIS
LIN {X -0.146,Y -455.165,Z 534.908,A 0.000,B 0.000,C 90.000,E1 19.450} C_DIS
LIN {X 0.055,Y -454.851,Z 534.899,A 0.000,B 0.000,C 90.000,E1 17.819} C_DIS
LIN {X -0.238,Y -454.555,Z 534.887,A 0.000,B 0.000,C 90.000,E1 15.607} C_DIS
LIN {X -0.220,Y -454.616,Z 534.874,A 0.000,B 0.000,C 90.000,E1 13.355} C_DIS
LIN {X -0.193,Y -455.108,Z 534.860,A 0.000,B 0.000,C 90.000,E1 10.782} C_DIS
LIN {X -0.017,Y -456.131,Z 534.844,A 0.000,B 0.000,C 90.000,E1 7.871} C_DIS
LIN {X -0.053,Y -457.622,Z 534.828,A 0.000,B 0.000,C 90.000,E1 4.992} C_DIS
LIN {X -0.024,Y -459.114,Z 534.815,A 0.000,B 0.000,C 90.000,E1 2.751} C_DIS
LIN {X -0.001,Y -460.987,Z 534.803,A 0.000,B 0.000,C 90.000,E1 0.516} C_DIS
LIN {X 0.062,Y -463.805,Z 534.788,A 0.000,B 0.000,C 90.000,E1 357.879} C_DIS
LIN {X -0.210,Y -467.336,Z 534.772,A 0.000,B 0.000,C 90.000,E1 355.065} C_DIS
LIN {X 0.141,Y -470.238,Z 534.760,A 0.000,B 0.000,C 90.000,E1 352.818} C_DIS
LIN {X -0.140,Y -472.796,Z 534.750,A 0.000,B 0.000,C 90.000,E1 350.971} C_DIS
LIN {X -0.054,Y -474.995,Z 534.741,A 0.000,B 0.000,C 90.000,E1 349.398} C_DIS
LIN {X -0.160,Y -480.408,Z 534.722,A 0.000,B 0.000,C 90.000,E1 345.992} C_DIS
LIN {X 0.001,Y -484.994,Z 534.708,A 0.000,B 0.000,C 90.000,E1 343.504} C_DIS
LIN {X 0.084,Y -489.181,Z 534.696,A 0.000,B 0.000,C 90.000,E1 341.348} C_DIS
LIN {X 0.091,Y -492.815,Z 534.686,A 0.000,B 0.000,C 90.000,E1 339.518} C_DIS
LIN {X -0.149,Y -495.816,Z 534.678,A 0.000,B 0.000,C 90.000,E1 338.028} C_DIS
LIN {X 0.131,Y -498.767,Z 534.669,A 0.000,B 0.000,C 90.000,E1 336.485} C_DIS
LIN {X 0.136,Y -501.103,Z 534.663,A 0.000,B 0.000,C 90.000,E1 335.281} C_DIS
LIN {X 0.256,Y -503.878,Z 534.654,A 0.000,B 0.000,C 90.000,E1 333.768} C_DIS
LIN {X -0.174,Y -507.209,Z 534.645,A 0.000,B 0.000,C 90.000,E1 332.025} C_DIS
LIN {X 0.151,Y -510.409,Z 534.635,A 0.000,B 0.000,C 90.000,E1 330.205} C_DIS
LIN {X 0.268,Y -514.213,Z 534.623,A 0.000,B 0.000,C 90.000,E1 328.122} C_DIS
LIN {X 0.047,Y -518.092,Z 534.612,A 0.000,B 0.000,C 90.000,E1 326.087} C_DIS
LIN {X 0.180,Y -520.851,Z 534.604,A 0.000,B 0.000,C 90.000,E1 324.609} C_DIS
LIN {X 0.323,Y -524.050,Z 534.594,A 0.000,B 0.000,C 90.000,E1 322.844} C_DIS
LIN {X 0.139,Y -526.842,Z 534.586,A 0.000,B 0.000,C 90.000,E1 321.412} C_DIS
LIN {X -0.107,Y -530.150,Z 534.576,A 0.000,B 0.000,C 90.000,E1 319.703} C_DIS
LIN {X 0.064,Y -533.760,Z 534.567,A 0.000,B 0.000,C 90.000,E1 317.957} C_DIS
LIN {X 0.246,Y -538.679,Z 534.554,A 0.000,B 0.000,C 90.000,E1 315.648} C_DIS
LIN {X 0.192,Y -543.836,Z 534.541,A 0.000,B 0.000,C 90.000,E1 313.380} C_DIS
LIN {X -0.128,Y -547.266,Z 534.533,A 0.000,B 0.000,C 90.000,E1 312.000} C_DIS
LIN {X -0.031,Y -550.656,Z 534.526,A 0.000,B 0.000,C 90.000,E1 310.583} C_DIS
LIN {X -0.236,Y -553.078,Z 534.519,A 0.000,B 0.000,C 90.000,E1 309.483} C_DIS
LIN {X -0.330,Y -556.023,Z 534.512,A 0.000,B 0.000,C 90.000,E1 308.096} C_DIS
LIN {X -0.013,Y -558.482,Z 534.505,A 0.000,B 0.000,C 90.000,E1 306.950} C_DIS
LIN {X -0.087,Y -560.821,Z 534.500,A 0.000,B 0.000,C 90.000,E1 306.091} C_DIS
LIN {X -0.110,Y -562.148,Z 534.499,A 0.000,B 0.000,C 90.000,E1 305.851} C_DIS
LIN {X -0.341,Y -563.353,Z 534.498,A 0.000,B 0.000,C 90.000,E1 305.598} C_DIS
LIN {X -0.239,Y -565.336,Z 534.496,A 0.000,B 0.000,C 90.000,E1 305.311} C_DIS
LIN {X -0.132,Y -566.854,Z 534.495,A 0.000,B 0.000,C 90.000,E1 305.025} C_DIS
LIN {X -0.011,Y -569.273,Z 534.493,A 0.000,B 0.000,C 90.000,E1 304.692} C_DIS
LIN {X 0.209,Y -570.195,Z 534.492,A 0.000,B 0.000,C 90.000,E1 304.532} C_DIS
LIN {X 0.200,Y -572.106,Z 534.491,A 0.000,B 0.000,C 90.000,E1 304.326} C_DIS
LIN {X 0.277,Y -575.281,Z 534.489,A 0.000,B 0.000,C 90.000,E1 303.913} C_DIS
LIN {X -0.035,Y -587.237,Z 534.481,A 0.000,B 0.000,C 90.000,E1 302.594} C_DIS
LIN {X -0.202,Y -596.764,Z 534.475,A 0.000,B 0.000,C 90.000,E1 301.544} C_DIS
LIN {X 0.153,Y -603.696,Z 534.471,A 0.000,B 0.000,C 90.000,E1 300.718} C_DIS
LIN {X 0.020,Y -608.023,Z 534.468,A 0.000,B 0.000,C 90.000,E1 300.207} C_DIS
LIN {X 0.246,Y -611.013,Z 534.466,A 0.000,B 0.000,C 90.000,E1 299.795} C_DIS
LIN {X 0.154,Y -615.660,Z 534.462,A 0.000,B 0.000,C 90.000,E1 299.155} C_DIS
LIN {X 0.119,Y -618.227,Z 534.460,A 0.000,B 0.000,C 90.000,E1 298.771} C_DIS
LIN {X -0.160,Y -621.927,Z 534.456,A 0.000,B 0.000,C 90.000,E1 298.153} C_DIS
LIN {X -0.163,Y -622.583,Z 534.456,A 0.000,B 0.000,C 90.000,E1 298.025} C_DIS
LIN {X -0.156,Y -625.578,Z 534.451,A 0.000,B 0.000,C 90.000,E1 297.257} C_DIS
LIN {X -0.147,Y -626.199,Z 534.450,A 0.000,B 0.000,C 90.000,E1 297.001} C_DIS
LIN {X -0.119,Y -626.980,Z 534.447,A 0.000,B 0.000,C 90.000,E1 296.488} C_DIS
LIN {X -0.103,Y -627.175,Z 534.446,A 0.000,B 0.000,C 90.000,E1 296.232} C_DIS
LIN {X -0.067,Y -627.098,Z 534.443,A 0.000,B 0.000,C 90.000,E1 295.720} C_DIS
LIN {X -0.032,Y -626.031,Z 534.440,A 0.000,B 0.000,C 90.000,E1 295.207} C_DIS
LIN {X -0.017,Y -625.284,Z 534.439,A 0.000,B 0.000,C 90.000,E1 294.951} C_DIS
LIN {X -0.257,Y -622.494,Z 534.436,A 0.000,B 0.000,C 90.000,E1 294.463} C_DIS
LIN {X -0.253,Y -619.239,Z 534.434,A 0.000,B 0.000,C 90.000,E1 294.079} C_DIS
LIN {X -0.241,Y -616.587,Z 534.432,A 0.000,B 0.000,C 90.000,E1 293.823} C_DIS
LIN {X 0.024,Y -612.671,Z 534.431,A 0.000,B 0.000,C 90.000,E1 293.590} C_DIS
LIN {X -0.041,Y -611.436,Z 534.431,A 0.000,B 0.000,C 90.000,E1 293.515} C_DIS
LIN {X -0.083,Y -610.597,Z 534.430,A 0.000,B 0.000,C 90.000,E1 293.439} C_DIS
LIN {X -0.271,Y -608.599,Z 534.430,A 0.000,B 0.000,C 90.000,E1 293.334} C_DIS
LIN {X -0.215,Y -605.567,Z 534.429,A 0.000,B 0.000,C 90.000,E1 293.206} C_DIS
LIN {X -0.103,Y -602.878,Z 534.428,A 0.000,B 0.000,C 90.000,E1 293.025} C_DIS
LIN {X 0.228,Y -601.092,Z 534.427,A 0.000,B 0.000,C 90.000,E1 292.898} C_DIS
LIN {X 0.186,Y -593.422,Z 534.426,A 0.000,B 0.000,C 90.000,E1 292.589} C_DIS
LIN {X 0.053,Y -589.819,Z 534.425,A 0.000,B 0.000,C 90.000,E1 292.461} C_DIS
LIN {X -0.068,Y -584.781,Z 534.424,A 0.000,B 0.000,C 90.000,E1 292.259} C_DIS
LIN {X 0.348,Y -578.606,Z 534.422,A 0.000,B 0.000,C 90.000,E1 291.897} C_DIS
LIN {X 0.042,Y -577.461,Z 534.421,A 0.000,B 0.000,C 90.000,E1 291.844} C_DIS
LIN {X -0.090,Y -574.999,Z 534.420,A 0.000,B 0.000,C 90.000,E1 291.642} C_DIS
LIN {X 0.071,Y -574.235,Z 534.419,A 0.000,B 0.000,C 90.000,E1 291.461} C_DIS
LIN {X -0.164,Y -573.904,Z 534.417,A 0.000,B 0.000,C 90.000,E1 291.153} C_DIS
LIN {X 0.191,Y -573.761,Z 534.413,A 0.000,B 0.000,C 90.000,E1 290.301} C_DIS
LIN {X 0.180,Y -574.038,Z 534.407,A 0.000,B 0.000,C 90.000,E1 289.214} C_DIS
LIN {X 0.176,Y -574.009,Z 534.401,A 0.000,B 0.000,C 90.000,E1 288.127} C_DIS
LIN {X 0.170,Y -573.905,Z 534.395,A 0.000,B 0.000,C 90.000,E1 287.040} C_DIS
LIN {X -0.005,Y -573.660,Z 534.389,A 0.000,B 0.000,C 90.000,E1 285.969} C_DIS
LIN {X -0.007,Y -572.871,Z 534.378,A 0.000,B 0.000,C 90.000,E1 284.064} C_DIS
LIN {X -0.015,Y -572.294,Z 534.371,A 0.000,B 0.000,C 90.000,E1 282.703} C_DIS
LIN {X -0.278,Y -571.676,Z 534.363,A 0.000,B 0.000,C 90.000,E1 281.366} C_DIS
LIN {X -0.153,Y -570.759,Z 534.352,A 0.000,B 0.000,C 90.000,E1 279.443} C_DIS
LIN {X -0.250,Y -570.018,Z 534.343,A 0.000,B 0.000,C 90.000,E1 277.814} C_DIS
LIN {X 0.217,Y -569.281,Z 534.333,A 0.000,B 0.000,C 90.000,E1 275.853} C_DIS
LIN {X 0.213,Y -568.921,Z 534.327,A 0.000,B 0.000,C 90.000,E1 274.759} C_DIS
LIN {X -0.289,Y -568.201,Z 534.319,A 0.000,B 0.000,C 90.000,E1 273.440} C_DIS
LIN {X -0.227,Y -567.381,Z 534.311,A 0.000,B 0.000,C 90.000,E1 272.064} C_DIS
LIN {X 0.266,Y -566.690,Z 534.305,A 0.000,B 0.000,C 90.000,E1 270.917} C_DIS
LIN {X -0.281,Y -565.668,Z 534.298,A 0.000,B 0.000,C 90.000,E1 269.599} C_DIS
LIN {X -0.157,Y -564.358,Z 534.289,A 0.000,B 0.000,C 90.000,E1 267.936} C_DIS
LIN {X 0.036,Y -562.858,Z 534.278,A 0.000,B 0.000,C 90.000,E1 265.988} C_DIS
LIN {X -0.152,Y -562.241,Z 534.273,A 0.000,B 0.000,C 90.000,E1 265.179} C_DIS
LIN {X -0.161,Y -561.014,Z 534.266,A 0.000,B 0.000,C 90.000,E1 263.799} C_DIS
LIN {X -0.067,Y -559.473,Z 534.256,A 0.000,B 0.000,C 90.000,E1 262.129} C_DIS
LIN {X -0.136,Y -558.423,Z 534.250,A 0.000,B 0.000,C 90.000,E1 261.027} C_DIS
LIN {X -0.083,Y -556.740,Z 534.242,A 0.000,B 0.000,C 90.000,E1 259.634} C_DIS
LIN {X 0.173,Y -554.688,Z 534.233,A 0.000,B 0.000,C 90.000,E1 257.937} C_DIS
LIN {X -0.280,Y -552.810,Z 534.225,A 0.000,B 0.000,C 90.000,E1 256.589} C_DIS
LIN {X -0.103,Y -550.711,Z 534.218,A 0.000,B 0.000,C 90.000,E1 255.172} C_DIS
LIN {X -0.252,Y -547.994,Z 534.208,A 0.000,B 0.000,C 90.000,E1 253.504} C_DIS
LIN {X -0.103,Y -545.926,Z 534.202,A 0.000,B 0.000,C 90.000,E1 252.362} C_DIS
LIN {X 0.255,Y -543.175,Z 534.194,A 0.000,B 0.000,C 90.000,E1 250.913} C_DIS
LIN {X 0.047,Y -540.268,Z 534.186,A 0.000,B 0.000,C 90.000,E1 249.518} C_DIS
LIN {X -0.028,Y -537.168,Z 534.178,A 0.000,B 0.000,C 90.000,E1 248.103} C_DIS
LIN {X 0.122,Y -535.229,Z 534.174,A 0.000,B 0.000,C 90.000,E1 247.230} C_DIS
LIN {X -0.034,Y -532.489,Z 534.167,A 0.000,B 0.000,C 90.000,E1 246.102} C_DIS
LIN {X -0.227,Y -529.574,Z 534.161,A 0.000,B 0.000,C 90.000,E1 244.973} C_DIS
LIN {X -0.069,Y -525.733,Z 534.153,A 0.000,B 0.000,C 90.000,E1 243.512} C_DIS
LIN {X 0.251,Y -521.681,Z 534.145,A 0.000,B 0.000,C 90.000,E1 242.025} C_DIS
LIN {X 0.114,Y -518.447,Z 534.138,A 0.000,B 0.000,C 90.000,E1 240.873} C_DIS
LIN {X -0.271,Y -515.158,Z 534.132,A 0.000,B 0.000,C 90.000,E1 239.744} C_DIS
LIN {X 0.007,Y -511.727,Z 534.125,A 0.000,B 0.000,C 90.000,E1 238.535} C_DIS
LIN {X 0.131,Y -507.297,Z 534.117,A 0.000,B 0.000,C 90.000,E1 237.041} C_DIS
LIN {X -0.250,Y -502.770,Z 534.109,A 0.000,B 0.000,C 90.000,E1 235.595} C_DIS
LIN {X 0.023,Y -496.691,Z 534.097,A 0.000,B 0.000,C 90.000,E1 233.463} C_DIS
LIN {X -0.109,Y -491.600,Z 534.087,A 0.000,B 0.000,C 90.000,E1 231.662} C_DIS
LIN {X -0.084,Y -484.945,Z 534.073,A 0.000,B 0.000,C 90.000,E1 229.218} C_DIS
LIN {X -0.240,Y -480.135,Z 534.063,A 0.000,B 0.000,C 90.000,E1 227.391} C_DIS
LIN {X 0.247,Y -474.680,Z 534.051,A 0.000,B 0.000,C 90.000,E1 225.162} C_DIS
LIN {X 0.070,Y -470.884,Z 534.042,A 0.000,B 0.000,C 90.000,E1 223.623} C_DIS
LIN {X -0.158,Y -467.210,Z 534.034,A 0.000,B 0.000,C 90.000,E1 222.081} C_DIS
LIN {X 0.200,Y -463.578,Z 534.025,A 0.000,B 0.000,C 90.000,E1 220.458} C_DIS
LIN {X 0.018,Y -458.583,Z 534.013,A 0.000,B 0.000,C 90.000,E1 218.257} C_DIS
LIN {X -0.024,Y -455.122,Z 534.004,A 0.000,B 0.000,C 90.000,E1 216.664} C_DIS
LIN {X 0.107,Y -449.729,Z 533.989,A 0.000,B 0.000,C 90.000,E1 214.072} C_DIS
LIN {X 0.055,Y -445.848,Z 533.979,A 0.000,B 0.000,C 90.000,E1 212.133} C_DIS
LIN {X -0.183,Y -442.128,Z 533.968,A 0.000,B 0.000,C 90.000,E1 210.207} C_DIS
LIN {X -0.121,Y -438.546,Z 533.957,A 0.000,B 0.000,C 90.000,E1 208.231} C_DIS
LIN {X 0.032,Y -435.153,Z 533.946,A 0.000,B 0.000,C 90.000,E1 206.232} C_DIS
LIN {X 0.119,Y -431.308,Z 533.933,A 0.000,B 0.000,C 90.000,E1 203.898} C_DIS
LIN {X -0.076,Y -427.696,Z 533.920,A 0.000,B 0.000,C 90.000,E1 201.589} C_DIS
LIN {X 0.092,Y -423.465,Z 533.903,A 0.000,B 0.000,C 90.000,E1 198.544} C_DIS
LIN {X -0.098,Y -420.507,Z 533.890,A 0.000,B 0.000,C 90.000,E1 196.205} C_DIS
LIN {X 0.111,Y -418.470,Z 533.881,A 0.000,B 0.000,C 90.000,E1 194.481} C_DIS
LIN {X 0.121,Y -416.793,Z 533.873,A 0.000,B 0.000,C 90.000,E1 193.119} C_DIS
LIN {X 0.150,Y -413.950,Z 533.860,A 0.000,B 0.000,C 90.000,E1 190.725} C_DIS
LIN {X 0.060,Y -411.664,Z 533.848,A 0.000,B 0.000,C 90.000,E1 188.681} C_DIS
LIN {X 0.133,Y -409.457,Z 533.837,A 0.000,B 0.000,C 90.000,E1 186.606} C_DIS
LIN {X 0.117,Y -406.481,Z 533.820,A 0.000,B 0.000,C 90.000,E1 183.498} C_DIS
LIN {X -0.052,Y -404.266,Z 533.804,A 0.000,B 0.000,C 90.000,E1 180.745} C_DIS
LIN {X 0.106,Y -402.646,Z 533.789,A 0.000,B 0.000,C 90.000,E1 177.936} C_DIS
LIN {X -0.194,Y -401.500,Z 533.771,A 0.000,B 0.000,C 90.000,E1 174.837} C_DIS
LIN {X 0.019,Y -401.001,Z 533.754,A 0.000,B 0.000,C 90.000,E1 171.659} C_DIS
LIN {X -0.091,Y -400.981,Z 533.744,A 0.000,B 0.000,C 90.000,E1 169.926} C_DIS
LIN {X -0.007,Y -401.247,Z 533.730,A 0.000,B 0.000,C 90.000,E1 167.465} C_DIS
LIN {X -0.122,Y -401.890,Z 533.715,A 0.000,B 0.000,C 90.000,E1 164.685} C_DIS
LIN {X -0.091,Y -402.798,Z 533.701,A 0.000,B 0.000,C 90.000,E1 162.236} C_DIS
LIN {X 0.113,Y -403.798,Z 533.690,A 0.000,B 0.000,C 90.000,E1 160.115} C_DIS
LIN {X 0.101,Y -404.989,Z 533.678,A 0.000,B 0.000,C 90.000,E1 158.028} C_DIS
LIN {X 0.003,Y -406.061,Z 533.668,A 0.000,B 0.000,C 90.000,E1 156.305} C_DIS
LIN {X -0.028,Y -407.492,Z 533.657,A 0.000,B 0.000,C 90.000,E1 154.229} C_DIS
LIN {X -0.217,Y -408.472,Z 533.649,A 0.000,B 0.000,C 90.000,E1 152.871} C_DIS
LIN {X -0.110,Y -409.633,Z 533.640,A 0.000,B 0.000,C 90.000,E1 151.129} C_DIS
LIN {X -0.143,Y -410.691,Z 533.630,A 0.000,B 0.000,C 90.000,E1 149.410} C_DIS
LIN {X -0.015,Y -411.692,Z 533.619,A 0.000,B 0.000,C 90.000,E1 147.327} C_DIS
LIN {X 0.082,Y -412.445,Z 533.609,A 0.000,B 0.000,C 90.000,E1 145.595} C_DIS
LIN {X -0.068,Y -412.912,Z 533.601,A 0.000,B 0.000,C 90.000,E1 144.242} C_DIS
LIN {X 0.045,Y -413.483,Z 533.592,A 0.000,B 0.000,C 90.000,E1 142.512} C_DIS
LIN {X 0.008,Y -413.845,Z 533.582,A 0.000,B 0.000,C 90.000,E1 140.803} C_DIS
LIN {X -0.018,Y -414.123,Z 533.573,A 0.000,B 0.000,C 90.000,E1 139.094} C_DIS
LIN {X 0.088,Y -414.296,Z 533.561,A 0.000,B 0.000,C 90.000,E1 137.025} C_DIS
LIN {X 0.013,Y -414.381,Z 533.552,A 0.000,B 0.000,C 90.000,E1 135.324} C_DIS
LIN {X -0.058,Y -414.397,Z 533.542,A 0.000,B 0.000,C 90.000,E1 133.623} C_DIS
LIN {X 0.021,Y -414.280,Z 533.535,A 0.000,B 0.000,C 90.000,E1 132.243} C_DIS
LIN {X -0.074,Y -414.119,Z 533.529,A 0.000,B 0.000,C 90.000,E1 131.229} C_DIS
LIN {X 0.138,Y -413.833,Z 533.523,A 0.000,B 0.000,C 90.000,E1 130.172} C_DIS
LIN {X -0.237,Y -413.377,Z 533.518,A 0.000,B 0.000,C 90.000,E1 129.197} C_DIS
LIN {X 0.046,Y -412.406,Z 533.508,A 0.000,B 0.000,C 90.000,E1 127.443} C_DIS
LIN {X 0.099,Y -412.165,Z 533.506,A 0.000,B 0.000,C 90.000,E1 127.076} C_DIS
LIN {X 0.060,Y -412.170,Z 533.506,A 0.000,B 0.000,C 90.000,E1 127.076} C_DIS
LIN {X -0.103,Y -415.207,Z 533.500,A 0.000,B 0.000,C 90.000,E1 126.091} C_DIS
LIN {X 0.008,Y -416.878,Z 533.497,A 0.000,B 0.000,C 90.000,E1 125.391} C_DIS
LIN {X -0.064,Y -426.598,Z 533.476,A 0.000,B 0.000,C 90.000,E1 121.671} C_DIS
LIN {X -0.101,Y -430.665,Z 533.469,A 0.000,B 0.000,C 90.000,E1 120.335} C_DIS
LIN {X -0.139,Y -440.629,Z 533.446,A 0.000,B 0.000,C 90.000,E1 116.360} C_DIS
LIN {X 0.019,Y -444.484,Z 533.439,A 0.000,B 0.000,C 90.000,E1 115.027} C_DIS
LIN {X -0.083,Y -445.945,Z 533.435,A 0.000,B 0.000,C 90.000,E1 114.387} C_DIS
LIN {X -0.059,Y -449.126,Z 533.427,A 0.000,B 0.000,C 90.000,E1 112.950} C_DIS
LIN {X -0.099,Y -449.187,Z 533.427,A 0.000,B 0.000,C 90.000,E1 112.950} C_DIS
LIN {X 0.255,Y -474.961,Z 533.422,A 0.000,B 0.000,C 90.000,E1 111.897} C_DIS
LIN {X -0.066,Y -485.538,Z 533.420,A 0.000,B 0.000,C 90.000,E1 111.535} C_DIS
LIN {X -0.040,Y -502.434,Z 533.416,A 0.000,B 0.000,C 90.000,E1 110.844} C_DIS
LIN {X 0.004,Y -509.238,Z 533.414,A 0.000,B 0.000,C 90.000,E1 110.556} C_DIS
LIN {X 0.214,Y -522.824,Z 533.411,A 0.000,B 0.000,C 90.000,E1 109.939} C_DIS
LIN {X -0.081,Y -532.718,Z 533.408,A 0.000,B 0.000,C 90.000,E1 109.504} C_DIS
LIN {X -0.067,Y -540.875,Z 533.406,A 0.000,B 0.000,C 90.000,E1 109.087} C_DIS
LIN {X -0.125,Y -548.902,Z 533.404,A 0.000,B 0.000,C 90.000,E1 108.652} C_DIS
LIN {X 0.239,Y -554.928,Z 533.401,A 0.000,B 0.000,C 90.000,E1 108.236} C_DIS
LIN {X 0.073,Y -560.426,Z 533.399,A 0.000,B 0.000,C 90.000,E1 107.873} C_DIS
LIN {X 0.127,Y -565.833,Z 533.397,A 0.000,B 0.000,C 90.000,E1 107.457} C_DIS
LIN {X 0.224,Y -571.205,Z 533.395,A 0.000,B 0.000,C 90.000,E1 106.985} C_DIS
LIN {X 0.031,Y -577.154,Z 533.391,A 0.000,B 0.000,C 90.000,E1 106.441} C_DIS
LIN {X 0.142,Y -581.605,Z 533.389,A 0.000,B 0.000,C 90.000,E1 105.969} C_DIS
LIN {X 0.000,Y -587.442,Z 533.385,A 0.000,B 0.000,C 90.000,E1 105.315} C_DIS
LIN {X 0.082,Y -591.722,Z 533.382,A 0.000,B 0.000,C 90.000,E1 104.773} C_DIS
LIN {X -0.004,Y -597.346,Z 533.378,A 0.000,B 0.000,C 90.000,E1 104.008} C_DIS
LIN {X -0.145,Y -602.756,Z 533.373,A 0.000,B 0.000,C 90.000,E1 103.231} C_DIS
LIN {X -0.270,Y -607.090,Z 533.370,A 0.000,B 0.000,C 90.000,E1 102.591} C_DIS
LIN {X -0.188,Y -611.906,Z 533.366,A 0.000,B 0.000,C 90.000,E1 101.827} C_DIS
LIN {X 0.115,Y -615.632,Z 533.362,A 0.000,B 0.000,C 90.000,E1 101.186} C_DIS
LIN {X -0.108,Y -619.919,Z 533.358,A 0.000,B 0.000,C 90.000,E1 100.433} C_DIS
LIN {X -0.176,Y -623.818,Z 533.354,A 0.000,B 0.000,C 90.000,E1 99.670} C_DIS
LIN {X 0.088,Y -628.653,Z 533.348,A 0.000,B 0.000,C 90.000,E1 98.624} C_DIS
LIN {X -0.009,Y -632.115,Z 533.344,A 0.000,B 0.000,C 90.000,E1 97.871} C_DIS
LIN {X 0.006,Y -637.749,Z 533.337,A 0.000,B 0.000,C 90.000,E1 96.606} C_DIS
LIN {X -0.006,Y -641.031,Z 533.333,A 0.000,B 0.000,C 90.000,E1 95.853} C_DIS
LIN {X -0.054,Y -644.013,Z 533.328,A 0.000,B 0.000,C 90.000,E1 95.106} C_DIS
LIN {X 0.164,Y -645.919,Z 533.326,A 0.000,B 0.000,C 90.000,E1 94.588} C_DIS
LIN {X -0.299,Y -647.661,Z 533.323,A 0.000,B 0.000,C 90.000,E1 94.131} C_DIS
LIN {X 0.190,Y -650.738,Z 533.317,A 0.000,B 0.000,C 90.000,E1 93.094} C_DIS
LIN {X -0.238,Y -652.070,Z 533.315,A 0.000,B 0.000,C 90.000,E1 92.636} C_DIS
LIN {X -0.204,Y -653.815,Z 533.310,A 0.000,B 0.000,C 90.000,E1 91.892} C_DIS
LIN {X -0.133,Y -655.143,Z 533.306,A 0.000,B 0.000,C 90.000,E1 91.146} C_DIS
LIN {X -0.066,Y -655.999,Z 533.302,A 0.000,B 0.000,C 90.000,E1 90.401} C_DIS
LIN {X 0.205,Y -656.401,Z 533.299,A 0.000,B 0.000,C 90.000,E1 89.885} C_DIS
LIN {X -0.179,Y -656.624,Z 533.297,A 0.000,B 0.000,C 90.000,E1 89.427} C_DIS
LIN {X -0.098,Y -656.649,Z 533.293,A 0.000,B 0.000,C 90.000,E1 88.682} C_DIS
LIN {X 0.194,Y -656.484,Z 533.290,A 0.000,B 0.000,C 90.000,E1 88.165} C_DIS
LIN {X 0.272,Y -655.988,Z 533.286,A 0.000,B 0.000,C 90.000,E1 87.421} C_DIS
LIN {X -0.281,Y -655.140,Z 533.282,A 0.000,B 0.000,C 90.000,E1 86.731} C_DIS
LIN {X -0.025,Y -654.431,Z 533.279,A 0.000,B 0.000,C 90.000,E1 86.216} C_DIS
LIN {X -0.149,Y -652.439,Z 533.274,A 0.000,B 0.000,C 90.000,E1 85.241} C_DIS
LIN {X -0.025,Y -650.696,Z 533.269,A 0.000,B 0.000,C 90.000,E1 84.489} C_DIS
LIN {X 0.025,Y -648.658,Z 533.265,A 0.000,B 0.000,C 90.000,E1 83.742} C_DIS
LIN {X -0.113,Y -645.600,Z 533.260,A 0.000,B 0.000,C 90.000,E1 82.761} C_DIS
LIN {X -0.040,Y -642.876,Z 533.256,A 0.000,B 0.000,C 90.000,E1 82.008} C_DIS
LIN {X -0.258,Y -638.960,Z 533.250,A 0.000,B 0.000,C 90.000,E1 81.027} C_DIS
LIN {X 0.194,Y -634.555,Z 533.245,A 0.000,B 0.000,C 90.000,E1 79.982} C_DIS
LIN {X -0.053,Y -628.885,Z 533.238,A 0.000,B 0.000,C 90.000,E1 78.870} C_DIS
LIN {X 0.083,Y -624.365,Z 533.233,A 0.000,B 0.000,C 90.000,E1 77.993} C_DIS
LIN {X 0.057,Y -619.992,Z 533.229,A 0.000,B 0.000,C 90.000,E1 77.229} C_DIS
LIN {X -0.012,Y -615.406,Z 533.225,A 0.000,B 0.000,C 90.000,E1 76.464} C_DIS
LIN {X -0.130,Y -610.137,Z 533.221,A 0.000,B 0.000,C 90.000,E1 75.700} C_DIS
LIN {X -0.096,Y -605.086,Z 533.217,A 0.000,B 0.000,C 90.000,E1 75.046} C_DIS
LIN {X -0.104,Y -599.446,Z 533.213,A 0.000,B 0.000,C 90.000,E1 74.393} C_DIS
LIN {X -0.090,Y -594.664,Z 533.210,A 0.000,B 0.000,C 90.000,E1 73.866} C_DIS
LIN {X 0.163,Y -589.525,Z 533.207,A 0.000,B 0.000,C 90.000,E1 73.323} C_DIS
LIN {X 0.008,Y -583.990,Z 533.205,A 0.000,B 0.000,C 90.000,E1 72.834} C_DIS
LIN {X -0.043,Y -578.223,Z 533.202,A 0.000,B 0.000,C 90.000,E1 72.362} C_DIS
LIN {X -0.114,Y -572.725,Z 533.200,A 0.000,B 0.000,C 90.000,E1 71.945} C_DIS
LIN {X 0.002,Y -566.766,Z 533.197,A 0.000,B 0.000,C 90.000,E1 71.511} C_DIS
LIN {X -0.223,Y -561.923,Z 533.196,A 0.000,B 0.000,C 90.000,E1 71.221} C_DIS
LIN {X 0.315,Y -555.340,Z 533.193,A 0.000,B 0.000,C 90.000,E1 70.786} C_DIS
LIN {X 0.178,Y -550.634,Z 533.192,A 0.000,B 0.000,C 90.000,E1 70.550} C_DIS
LIN {X -0.038,Y -545.087,Z 533.191,A 0.000,B 0.000,C 90.000,E1 70.315} C_DIS
LIN {X 0.218,Y -539.745,Z 533.189,A 0.000,B 0.000,C 90.000,E1 70.061} C_DIS
LIN {X -0.148,Y -532.417,Z 533.188,A 0.000,B 0.000,C 90.000,E1 69.826} C_DIS
LIN {X 0.195,Y -521.503,Z 533.186,A 0.000,B 0.000,C 90.000,E1 69.444} C_DIS
LIN {X -0.055,Y -512.734,Z 533.185,A 0.000,B 0.000,C 90.000,E1 69.209} C_DIS
LIN {X -0.018,Y -501.619,Z 533.183,A 0.000,B 0.000,C 90.000,E1 68.901} C_DIS
LIN {X 0.175,Y -492.210,Z 533.182,A 0.000,B 0.000,C 90.000,E1 68.646} C_DIS
LIN {X 0.070,Y -467.174,Z 533.178,A 0.000,B 0.000,C 90.000,E1 68.050} C_DIS
LIN {X 0.023,Y -467.035,Z 533.178,A 0.000,B 0.000,C 90.000,E1 68.050} C_DIS
LIN {X -0.225,Y -465.572,Z 533.172,A 0.000,B 0.000,C 90.000,E1 67.050} C_DIS
LIN {X 0.163,Y -457.114,Z 533.149,A 0.000,B 0.000,C 90.000,E1 62.871} C_DIS
LIN {X 0.272,Y -455.532,Z 533.144,A 0.000,B 0.000,C 90.000,E1 61.897} C_DIS
LIN {X 0.037,Y -445.587,Z 533.119,A 0.000,B 0.000,C 90.000,E1 57.406} C_DIS
LIN {X 0.086,Y -444.119,Z 533.114,A 0.000,B 0.000,C 90.000,E1 56.580} C_DIS
LIN {X 0.047,Y -444.114,Z 533.114,A 0.000,B 0.000,C 90.000,E1 56.580} C_DIS
LIN {X -0.105,Y -446.771,Z 533.108,A 0.000,B 0.000,C 90.000,E1 55.468} C_DIS
LIN {X -0.028,Y -448.946,Z 533.103,A 0.000,B 0.000,C 90.000,E1 54.482} C_DIS
LIN {X 0.127,Y -452.307,Z 533.094,A 0.000,B 0.000,C 90.000,E1 52.844} C_DIS
LIN {X 0.265,Y -454.693,Z 533.087,A 0.000,B 0.000,C 90.000,E1 51.537} C_DIS
LIN {X 0.085,Y -456.888,Z 533.079,A 0.000,B 0.000,C 90.000,E1 50.275} C_DIS
LIN {X 0.208,Y -458.383,Z 533.074,A 0.000,B 0.000,C 90.000,E1 49.299} C_DIS
LIN {X 0.113,Y -460.674,Z 533.065,A 0.000,B 0.000,C 90.000,E1 47.715} C_DIS
LIN {X -0.070,Y -461.780,Z 533.060,A 0.000,B 0.000,C 90.000,E1 46.782} C_DIS
LIN {X 0.077,Y -462.697,Z 533.055,A 0.000,B 0.000,C 90.000,E1 45.810} C_DIS
LIN {X -0.034,Y -463.572,Z 533.048,A 0.000,B 0.000,C 90.000,E1 44.555} C_DIS
LIN {X -0.188,Y -464.080,Z 533.042,A 0.000,B 0.000,C 90.000,E1 43.623} C_DIS
LIN {X 0.070,Y -464.566,Z 533.035,A 0.000,B 0.000,C 90.000,E1 42.324} C_DIS
LIN {X -0.065,Y -464.731,Z 533.030,A 0.000,B 0.000,C 90.000,E1 41.391} C_DIS
LIN {X 0.205,Y -464.665,Z 533.023,A 0.000,B 0.000,C 90.000,E1 40.092} C_DIS
LIN {X 0.171,Y -464.452,Z 533.016,A 0.000,B 0.000,C 90.000,E1 38.830} C_DIS
LIN {X -0.155,Y -464.096,Z 533.009,A 0.000,B 0.000,C 90.000,E1 37.604} C_DIS
LIN {X 0.165,Y -463.591,Z 533.002,A 0.000,B 0.000,C 90.000,E1 36.297} C_DIS
LIN {X -0.176,Y -462.561,Z 532.990,A 0.000,B 0.000,C 90.000,E1 34.119} C_DIS
LIN {X -0.035,Y -461.930,Z 532.982,A 0.000,B 0.000,C 90.000,E1 32.832} C_DIS
LIN {X -0.166,Y -461.147,Z 532.974,A 0.000,B 0.000,C 90.000,E1 31.258} C_DIS
LIN {X -0.038,Y -460.069,Z 532.963,A 0.000,B 0.000,C 90.000,E1 29.333} C_DIS
LIN {X 0.241,Y -458.985,Z 532.952,A 0.000,B 0.000,C 90.000,E1 27.385} C_DIS
LIN {X 0.286,Y -457.959,Z 532.942,A 0.000,B 0.000,C 90.000,E1 25.463} C_DIS
LIN {X 0.105,Y -457.043,Z 532.931,A 0.000,B 0.000,C 90.000,E1 23.567} C_DIS
LIN {X -0.034,Y -456.299,Z 532.920,A 0.000,B 0.000,C 90.000,E1 21.663} C_DIS
LIN {X 0.050,Y -455.462,Z 532.906,A 0.000,B 0.000,C 90.000,E1 19.087} C_DIS
LIN {X -0.072,Y -455.196,Z 532.899,A 0.000,B 0.000,C 90.000,E1 17.819} C_DIS
LIN {X -0.005,Y -454.939,Z 532.890,A 0.000,B 0.000,C 90.000,E1 16.205} C_DIS
LIN {X -0.097,Y -454.879,Z 532.876,A 0.000,B 0.000,C 90.000,E1 13.647} C_DIS
LIN {X -0.052,Y -455.156,Z 532.865,A 0.000,B 0.000,C 90.000,E1 11.715} C_DIS
LIN {X -0.082,Y -455.603,Z 532.854,A 0.000,B 0.000,C 90.000,E1 9.792} C_DIS
LIN {X -0.178,Y -456.629,Z 532.840,A 0.000,B 0.000,C 90.000,E1 7.239} C_DIS
LIN {X -0.191,Y -458.206,Z 532.824,A 0.000,B 0.000,C 90.000,E1 4.359} C_DIS
LIN {X -0.221,Y -460.308,Z 532.808,A 0.000,B 0.000,C 90.000,E1 1.489} C_DIS
LIN {X -0.164,Y -463.572,Z 532.790,A 0.000,B 0.000,C 90.000,E1 358.224} C_DIS
LIN {X -0.215,Y -466.601,Z 532.776,A 0.000,B 0.000,C 90.000,E1 355.698} C_DIS
LIN {X 0.039,Y -468.637,Z 532.767,A 0.000,B 0.000,C 90.000,E1 354.090} C_DIS
LIN {X 0.188,Y -471.165,Z 532.757,A 0.000,B 0.000,C 90.000,E1 352.186} C_DIS
LIN {X -0.005,Y -473.789,Z 532.746,A 0.000,B 0.000,C 90.000,E1 350.330} C_DIS
LIN {X -0.059,Y -476.453,Z 532.736,A 0.000,B 0.000,C 90.000,E1 348.465} C_DIS
LIN {X 0.177,Y -481.039,Z 532.720,A 0.000,B 0.000,C 90.000,E1 345.644} C_DIS
LIN {X 0.023,Y -485.699,Z 532.707,A 0.000,B 0.000,C 90.000,E1 343.196} C_DIS
LIN {X 0.130,Y -489.902,Z 532.695,A 0.000,B 0.000,C 90.000,E1 341.040} C_DIS
LIN {X 0.119,Y -492.942,Z 532.686,A 0.000,B 0.000,C 90.000,E1 339.518} C_DIS
LIN {X -0.118,Y -495.975,Z 532.678,A 0.000,B 0.000,C 90.000,E1 338.028} C_DIS
LIN {X -0.232,Y -499.519,Z 532.668,A 0.000,B 0.000,C 90.000,E1 336.230} C_DIS
LIN {X -0.142,Y -502.374,Z 532.659,A 0.000,B 0.000,C 90.000,E1 334.717} C_DIS
LIN {X -0.008,Y -505.168,Z 532.651,A 0.000,B 0.000,C 90.000,E1 333.204} C_DIS
LIN {X -0.052,Y -507.939,Z 532.643,A 0.000,B 0.000,C 90.000,E1 331.719} C_DIS
LIN {X 0.093,Y -511.150,Z 532.633,A 0.000,B 0.000,C 90.000,E1 329.921} C_DIS
LIN {X 0.050,Y -514.453,Z 532.623,A 0.000,B 0.000,C 90.000,E1 328.152} C_DIS
LIN {X 0.108,Y -518.353,Z 532.612,A 0.000,B 0.000,C 90.000,E1 326.087} C_DIS
LIN {X -0.109,Y -521.660,Z 532.602,A 0.000,B 0.000,C 90.000,E1 324.356} C_DIS
LIN {X -0.061,Y -524.900,Z 532.592,A 0.000,B 0.000,C 90.000,E1 322.603} C_DIS
LIN {X -0.195,Y -527.166,Z 532.586,A 0.000,B 0.000,C 90.000,E1 321.457} C_DIS
LIN {X -0.021,Y -530.468,Z 532.576,A 0.000,B 0.000,C 90.000,E1 319.703} C_DIS
LIN {X 0.174,Y -533.470,Z 532.568,A 0.000,B 0.000,C 90.000,E1 318.243} C_DIS
LIN {X -0.005,Y -537.692,Z 532.557,A 0.000,B 0.000,C 90.000,E1 316.257} C_DIS
LIN {X -0.065,Y -540.795,Z 532.549,A 0.000,B 0.000,C 90.000,E1 314.838} C_DIS
LIN {X 0.334,Y -546.028,Z 532.536,A 0.000,B 0.000,C 90.000,E1 312.528} C_DIS
LIN {X 0.097,Y -550.079,Z 532.527,A 0.000,B 0.000,C 90.000,E1 310.862} C_DIS
LIN {X 0.249,Y -552.627,Z 532.521,A 0.000,B 0.000,C 90.000,E1 309.725} C_DIS
LIN {X -0.282,Y -555.526,Z 532.513,A 0.000,B 0.000,C 90.000,E1 308.382} C_DIS
LIN {X 0.197,Y -559.145,Z 532.504,A 0.000,B 0.000,C 90.000,E1 306.664} C_DIS
LIN {X -0.196,Y -560.909,Z 532.500,A 0.000,B 0.000,C 90.000,E1 306.011} C_DIS
LIN {X 0.107,Y -562.294,Z 532.498,A 0.000,B 0.000,C 90.000,E1 305.644} C_DIS
LIN {X -0.122,Y -563.227,Z 532.497,A 0.000,B 0.000,C 90.000,E1 305.391} C_DIS
LIN {X 0.193,Y -565.266,Z 532.494,A 0.000,B 0.000,C 90.000,E1 304.945} C_DIS
LIN {X -0.327,Y -569.200,Z 532.491,A 0.000,B 0.000,C 90.000,E1 304.405} C_DIS
LIN {X -0.206,Y -571.403,Z 532.490,A 0.000,B 0.000,C 90.000,E1 304.119} C_DIS
LIN {X -0.303,Y -572.284,Z 532.489,A 0.000,B 0.000,C 90.000,E1 303.992} C_DIS
LIN {X 0.364,Y -577.225,Z 532.485,A 0.000,B 0.000,C 90.000,E1 303.293} C_DIS
LIN {X -0.139,Y -593.113,Z 532.475,A 0.000,B 0.000,C 90.000,E1 301.514} C_DIS
LIN {X -0.037,Y -601.143,Z 532.470,A 0.000,B 0.000,C 90.000,E1 300.590} C_DIS
LIN {X -0.155,Y -604.269,Z 532.468,A 0.000,B 0.000,C 90.000,E1 300.207} C_DIS
LIN {X -0.077,Y -611.805,Z 532.462,A 0.000,B 0.000,C 90.000,E1 299.155} C_DIS
LIN {X 0.122,Y -616.739,Z 532.458,A 0.000,B 0.000,C 90.000,E1 298.359} C_DIS
LIN {X 0.087,Y -619.405,Z 532.455,A 0.000,B 0.000,C 90.000,E1 297.847} C_DIS
LIN {X 0.078,Y -620.556,Z 532.453,A 0.000,B 0.000,C 90.000,E1 297.590} C_DIS
LIN {X 0.071,Y -621.565,Z 532.452,A 0.000,B 0.000,C 90.000,E1 297.334} C_DIS
LIN {X 0.069,Y -622.976,Z 532.449,A 0.000,B 0.000,C 90.000,E1 296.821} C_DIS
LIN {X 0.072,Y -623.401,Z 532.448,A 0.000,B 0.000,C 90.000,E1 296.565} C_DIS
LIN {X 0.092,Y -623.726,Z 532.443,A 0.000,B 0.000,C 90.000,E1 295.796} C_DIS
LIN {X 0.106,Y -622.979,Z 532.441,A 0.000,B 0.000,C 90.000,E1 295.283} C_DIS
LIN {X 0.111,Y -622.174,Z 532.439,A 0.000,B 0.000,C 90.000,E1 295.027} C_DIS
LIN {X 0.114,Y -620.640,Z 532.437,A 0.000,B 0.000,C 90.000,E1 294.643} C_DIS
LIN {X 0.113,Y -619.907,Z 532.436,A 0.000,B 0.000,C 90.000,E1 294.515} C_DIS
LIN {X 0.100,Y -616.589,Z 532.434,A 0.000,B 0.000,C 90.000,E1 294.131} C_DIS
LIN {X -0.157,Y -615.715,Z 532.433,A 0.000,B 0.000,C 90.000,E1 294.027} C_DIS
LIN {X -0.138,Y -614.222,Z 532.433,A 0.000,B 0.000,C 90.000,E1 293.898} C_DIS
LIN {X -0.118,Y -612.094,Z 532.432,A 0.000,B 0.000,C 90.000,E1 293.770} C_DIS
LIN {X -0.022,Y -608.644,Z 532.430,A 0.000,B 0.000,C 90.000,E1 293.462} C_DIS
LIN {X 0.051,Y -606.126,Z 532.430,A 0.000,B 0.000,C 90.000,E1 293.334} C_DIS
LIN {X 0.002,Y -601.155,Z 532.428,A 0.000,B 0.000,C 90.000,E1 293.025} C_DIS
LIN {X 0.096,Y -596.664,Z 532.427,A 0.000,B 0.000,C 90.000,E1 292.823} C_DIS
LIN {X 0.066,Y -584.968,Z 532.424,A 0.000,B 0.000,C 90.000,E1 292.333} C_DIS
LIN {X -0.164,Y -579.518,Z 532.423,A 0.000,B 0.000,C 90.000,E1 292.078} C_DIS
LIN {X 0.073,Y -578.410,Z 532.422,A 0.000,B 0.000,C 90.000,E1 291.972} C_DIS
LIN {X 0.251,Y -577.211,Z 532.422,A 0.000,B 0.000,C 90.000,E1 291.844} C_DIS
LIN {X -0.167,Y -575.664,Z 532.421,A 0.000,B 0.000,C 90.000,E1 291.716} C_DIS
LIN {X -0.209,Y -575.619,Z 532.421,A 0.000,B 0.000,C 90.000,E1 291.716} C_DIS
LIN {X 0.205,Y -575.027,Z 532.420,A 0.000,B 0.000,C 90.000,E1 291.535} C_DIS
LIN {X -0.104,Y -574.667,Z 532.417,A 0.000,B 0.000,C 90.000,E1 291.153} C_DIS
LIN {X 0.259,Y -574.634,Z 532.413,A 0.000,B 0.000,C 90.000,E1 290.301} C_DIS
LIN {X 0.084,Y -574.906,Z 532.408,A 0.000,B 0.000,C 90.000,E1 289.504} C_DIS
LIN {X 0.086,Y -574.966,Z 532.402,A 0.000,B 0.000,C 90.000,E1 288.417} C_DIS
LIN {X 0.277,Y -574.869,Z 532.395,A 0.000,B 0.000,C 90.000,E1 287.040} C_DIS
LIN {X -0.086,Y -574.520,Z 532.387,A 0.000,B 0.000,C 90.000,E1 285.717} C_DIS
LIN {X -0.221,Y -573.772,Z 532.377,A 0.000,B 0.000,C 90.000,E1 283.828} C_DIS
LIN {X -0.215,Y -573.215,Z 532.369,A 0.000,B 0.000,C 90.000,E1 282.467} C_DIS
LIN {X -0.100,Y -572.741,Z 532.363,A 0.000,B 0.000,C 90.000,E1 281.366} C_DIS
LIN {X 0.052,Y -571.885,Z 532.353,A 0.000,B 0.000,C 90.000,E1 279.443} C_DIS
LIN {X 0.273,Y -570.940,Z 532.340,A 0.000,B 0.000,C 90.000,E1 277.239} C_DIS
LIN {X -0.093,Y -570.414,Z 532.333,A 0.000,B 0.000,C 90.000,E1 275.910} C_DIS
LIN {X -0.129,Y -570.030,Z 532.327,A 0.000,B 0.000,C 90.000,E1 274.821} C_DIS
LIN {X 0.002,Y -569.320,Z 532.319,A 0.000,B 0.000,C 90.000,E1 273.440} C_DIS
LIN {X 0.084,Y -568.498,Z 532.312,A 0.000,B 0.000,C 90.000,E1 272.064} C_DIS
LIN {X 0.148,Y -567.567,Z 532.304,A 0.000,B 0.000,C 90.000,E1 270.688} C_DIS
LIN {X 0.064,Y -566.729,Z 532.298,A 0.000,B 0.000,C 90.000,E1 269.599} C_DIS
LIN {X 0.209,Y -565.386,Z 532.289,A 0.000,B 0.000,C 90.000,E1 267.936} C_DIS
LIN {X -0.136,Y -563.814,Z 532.278,A 0.000,B 0.000,C 90.000,E1 266.045} C_DIS
LIN {X -0.218,Y -562.934,Z 532.272,A 0.000,B 0.000,C 90.000,E1 264.951} C_DIS
LIN {X -0.220,Y -561.626,Z 532.264,A 0.000,B 0.000,C 90.000,E1 263.571} C_DIS
LIN {X -0.190,Y -560.257,Z 532.257,A 0.000,B 0.000,C 90.000,E1 262.186} C_DIS
LIN {X -0.246,Y -559.139,Z 532.250,A 0.000,B 0.000,C 90.000,E1 261.084} C_DIS
LIN {X -0.038,Y -557.110,Z 532.241,A 0.000,B 0.000,C 90.000,E1 259.398} C_DIS
LIN {X 0.229,Y -555.050,Z 532.232,A 0.000,B 0.000,C 90.000,E1 257.701} C_DIS
LIN {X -0.218,Y -553.095,Z 532.224,A 0.000,B 0.000,C 90.000,E1 256.353} C_DIS
LIN {X -0.036,Y -550.931,Z 532.216,A 0.000,B 0.000,C 90.000,E1 254.936} C_DIS
LIN {X 0.248,Y -548.623,Z 532.209,A 0.000,B 0.000,C 90.000,E1 253.504} C_DIS
LIN {X -0.117,Y -546.520,Z 532.202,A 0.000,B 0.000,C 90.000,E1 252.417} C_DIS
LIN {X -0.194,Y -543.140,Z 532.193,A 0.000,B 0.000,C 90.000,E1 250.732} C_DIS
LIN {X 0.293,Y -540.169,Z 532.185,A 0.000,B 0.000,C 90.000,E1 249.263} C_DIS
LIN {X -0.058,Y -536.351,Z 532.176,A 0.000,B 0.000,C 90.000,E1 247.592} C_DIS
LIN {X -0.203,Y -532.905,Z 532.168,A 0.000,B 0.000,C 90.000,E1 246.177} C_DIS
LIN {X 0.308,Y -529.974,Z 532.161,A 0.000,B 0.000,C 90.000,E1 244.973} C_DIS
LIN {X 0.000,Y -526.104,Z 532.153,A 0.000,B 0.000,C 90.000,E1 243.563} C_DIS
LIN {X 0.087,Y -522.050,Z 532.145,A 0.000,B 0.000,C 90.000,E1 242.103} C_DIS
LIN {X -0.125,Y -517.981,Z 532.137,A 0.000,B 0.000,C 90.000,E1 240.667} C_DIS
LIN {X -0.152,Y -513.813,Z 532.129,A 0.000,B 0.000,C 90.000,E1 239.203} C_DIS
LIN {X 0.075,Y -508.547,Z 532.119,A 0.000,B 0.000,C 90.000,E1 237.406} C_DIS
LIN {X -0.008,Y -504.007,Z 532.111,A 0.000,B 0.000,C 90.000,E1 235.928} C_DIS
LIN {X 0.147,Y -496.106,Z 532.096,A 0.000,B 0.000,C 90.000,E1 233.210} C_DIS
LIN {X -0.012,Y -491.010,Z 532.086,A 0.000,B 0.000,C 90.000,E1 231.412} C_DIS
LIN {X -0.216,Y -485.187,Z 532.074,A 0.000,B 0.000,C 90.000,E1 229.299} C_DIS
LIN {X 0.311,Y -480.364,Z 532.064,A 0.000,B 0.000,C 90.000,E1 227.391} C_DIS
LIN {X 0.127,Y -474.888,Z 532.052,A 0.000,B 0.000,C 90.000,E1 225.243} C_DIS
LIN {X 0.044,Y -470.300,Z 532.041,A 0.000,B 0.000,C 90.000,E1 223.380} C_DIS
LIN {X 0.045,Y -467.408,Z 532.034,A 0.000,B 0.000,C 90.000,E1 222.123} C_DIS
LIN {X -0.151,Y -463.023,Z 532.024,A 0.000,B 0.000,C 90.000,E1 220.253} C_DIS
LIN {X -0.077,Y -458.760,Z 532.013,A 0.000,B 0.000,C 90.000,E1 218.338} C_DIS
LIN {X -0.113,Y -455.298,Z 532.004,A 0.000,B 0.000,C 90.000,E1 216.744} C_DIS
LIN {X 0.281,Y -449.903,Z 531.990,A 0.000,B 0.000,C 90.000,E1 214.119} C_DIS
LIN {X -0.014,Y -446.018,Z 531.979,A 0.000,B 0.000,C 90.000,E1 212.212} C_DIS
LIN {X -0.019,Y -442.317,Z 531.968,A 0.000,B 0.000,C 90.000,E1 210.256} C_DIS
LIN {X 0.039,Y -438.721,Z 531.957,A 0.000,B 0.000,C 90.000,E1 208.281} C_DIS
LIN {X -0.005,Y -435.305,Z 531.946,A 0.000,B 0.000,C 90.000,E1 206.309} C_DIS
LIN {X 0.061,Y -433.098,Z 531.939,A 0.000,B 0.000,C 90.000,E1 204.975} C_DIS
LIN {X 0.091,Y -429.337,Z 531.926,A 0.000,B 0.000,C 90.000,E1 202.642} C_DIS
LIN {X 0.075,Y -426.831,Z 531.917,A 0.000,B 0.000,C 90.000,E1 200.972} C_DIS
LIN {X -0.113,Y -423.131,Z 531.902,A 0.000,B 0.000,C 90.000,E1 198.308} C_DIS
LIN {X -0.136,Y -419.839,Z 531.887,A 0.000,B 0.000,C 90.000,E1 195.607} C_DIS
LIN {X 0.108,Y -417.321,Z 531.875,A 0.000,B 0.000,C 90.000,E1 193.536} C_DIS
LIN {X -0.169,Y -414.440,Z 531.862,A 0.000,B 0.000,C 90.000,E1 191.186} C_DIS
LIN {X 0.053,Y -412.563,Z 531.853,A 0.000,B 0.000,C 90.000,E1 189.443} C_DIS
LIN {X -0.142,Y -410.342,Z 531.841,A 0.000,B 0.000,C 90.000,E1 187.409} C_DIS
LIN {X -0.100,Y -408.186,Z 531.830,A 0.000,B 0.000,C 90.000,E1 185.334} C_DIS
LIN {X -0.200,Y -405.709,Z 531.814,A 0.000,B 0.000,C 90.000,E1 182.579} C_DIS
LIN {X 0.088,Y -404.404,Z 531.805,A 0.000,B 0.000,C 90.000,E1 180.802} C_DIS
LIN {X -0.130,Y -402.946,Z 531.791,A 0.000,B 0.000,C 90.000,E1 178.396} C_DIS
LIN {X -0.046,Y -401.590,Z 531.772,A 0.000,B 0.000,C 90.000,E1 174.894} C_DIS
LIN {X 0.106,Y -401.110,Z 531.752,A 0.000,B 0.000,C 90.000,E1 171.376} C_DIS
LIN {X 0.105,Y -401.198,Z 531.737,A 0.000,B 0.000,C 90.000,E1 168.578} C_DIS
LIN {X 0.213,Y -401.550,Z 531.725,A 0.000,B 0.000,C 90.000,E1 166.464} C_DIS
LIN {X 0.102,Y -402.334,Z 531.709,A 0.000,B 0.000,C 90.000,E1 163.685} C_DIS
LIN {X 0.159,Y -403.214,Z 531.698,A 0.000,B 0.000,C 90.000,E1 161.583} C_DIS
LIN {X -0.116,Y -404.065,Z 531.688,A 0.000,B 0.000,C 90.000,E1 159.880} C_DIS
LIN {X 0.147,Y -405.092,Z 531.679,A 0.000,B 0.000,C 90.000,E1 158.103} C_DIS
LIN {X 0.208,Y -406.190,Z 531.669,A 0.000,B 0.000,C 90.000,E1 156.357} C_DIS
LIN {X 0.093,Y -407.879,Z 531.655,A 0.000,B 0.000,C 90.000,E1 153.948} C_DIS
LIN {X 0.094,Y -408.851,Z 531.648,A 0.000,B 0.000,C 90.000,E1 152.564} C_DIS
LIN {X 0.043,Y -409.989,Z 531.638,A 0.000,B 0.000,C 90.000,E1 150.845} C_DIS
LIN {X 0.098,Y -410.869,Z 531.630,A 0.000,B 0.000,C 90.000,E1 149.459} C_DIS
LIN {X 0.017,Y -411.906,Z 531.619,A 0.000,B 0.000,C 90.000,E1 147.406} C_DIS
LIN {X 0.115,Y -412.671,Z 531.609,A 0.000,B 0.000,C 90.000,E1 145.674} C_DIS
LIN {X -0.107,Y -413.318,Z 531.600,A 0.000,B 0.000,C 90.000,E1 143.989} C_DIS
LIN {X -0.071,Y -413.874,Z 531.590,A 0.000,B 0.000,C 90.000,E1 142.271} C_DIS
LIN {X -0.094,Y -414.263,Z 531.581,A 0.000,B 0.000,C 90.000,E1 140.561} C_DIS
LIN {X -0.108,Y -414.531,Z 531.571,A 0.000,B 0.000,C 90.000,E1 138.852} C_DIS
LIN {X -0.159,Y -414.696,Z 531.562,A 0.000,B 0.000,C 90.000,E1 137.148} C_DIS
LIN {X -0.054,Y -414.827,Z 531.550,A 0.000,B 0.000,C 90.000,E1 135.081} C_DIS
LIN {X 0.015,Y -414.824,Z 531.543,A 0.000,B 0.000,C 90.000,E1 133.704} C_DIS
LIN {X 0.099,Y -414.688,Z 531.535,A 0.000,B 0.000,C 90.000,E1 132.324} C_DIS
LIN {X 0.010,Y -414.486,Z 531.530,A 0.000,B 0.000,C 90.000,E1 131.310} C_DIS
LIN {X -0.088,Y -414.178,Z 531.524,A 0.000,B 0.000,C 90.000,E1 130.297} C_DIS
LIN {X -0.143,Y -413.714,Z 531.518,A 0.000,B 0.000,C 90.000,E1 129.277} C_DIS
LIN {X 0.149,Y -412.706,Z 531.509,A 0.000,B 0.000,C 90.000,E1 127.523} C_DIS
LIN {X -0.086,Y -412.367,Z 531.506,A 0.000,B 0.000,C 90.000,E1 127.030} C_DIS
LIN {X -0.124,Y -412.380,Z 531.506,A 0.000,B 0.000,C 90.000,E1 127.030} C_DIS
LIN {X 0.178,Y -415.885,Z 531.499,A 0.000,B 0.000,C 90.000,E1 125.804} C_DIS
LIN {X 0.061,Y -425.361,Z 531.478,A 0.000,B 0.000,C 90.000,E1 122.084} C_DIS
LIN {X 0.004,Y -430.375,Z 531.469,A 0.000,B 0.000,C 90.000,E1 120.413} C_DIS
LIN {X 0.009,Y -431.987,Z 531.465,A 0.000,B 0.000,C 90.000,E1 119.745} C_DIS
LIN {X 0.002,Y -441.306,Z 531.445,A 0.000,B 0.000,C 90.000,E1 116.104} C_DIS
LIN {X -0.273,Y -444.209,Z 531.440,A 0.000,B 0.000,C 90.000,E1 115.155} C_DIS
LIN {X 0.172,Y -445.083,Z 531.438,A 0.000,B 0.000,C 90.000,E1 114.771} C_DIS
LIN {X -0.116,Y -449.872,Z 531.426,A 0.000,B 0.000,C 90.000,E1 112.642} C_DIS
LIN {X -0.156,Y -449.910,Z 531.426,A 0.000,B 0.000,C 90.000,E1 112.642} C_DIS
LIN {X -0.028,Y -470.214,Z 531.421,A 0.000,B 0.000,C 90.000,E1 111.844} C_DIS
LIN {X 0.028,Y -487.798,Z 531.418,A 0.000,B 0.000,C 90.000,E1 111.173} C_DIS
LIN {X 0.022,Y -505.076,Z 531.414,A 0.000,B 0.000,C 90.000,E1 110.482} C_DIS
LIN {X -0.089,Y -515.101,Z 531.411,A 0.000,B 0.000,C 90.000,E1 110.066} C_DIS
LIN {X -0.107,Y -525.184,Z 531.409,A 0.000,B 0.000,C 90.000,E1 109.631} C_DIS
LIN {X 0.112,Y -535.058,Z 531.406,A 0.000,B 0.000,C 90.000,E1 109.141} C_DIS
LIN {X -0.107,Y -541.575,Z 531.405,A 0.000,B 0.000,C 90.000,E1 108.833} C_DIS
LIN {X -0.109,Y -548.078,Z 531.403,A 0.000,B 0.000,C 90.000,E1 108.489} C_DIS
LIN {X -0.166,Y -554.079,Z 531.401,A 0.000,B 0.000,C 90.000,E1 108.127} C_DIS
LIN {X 0.182,Y -560.013,Z 531.398,A 0.000,B 0.000,C 90.000,E1 107.692} C_DIS
LIN {X -0.124,Y -564.458,Z 531.397,A 0.000,B 0.000,C 90.000,E1 107.402} C_DIS
LIN {X 0.126,Y -571.351,Z 531.393,A 0.000,B 0.000,C 90.000,E1 106.804} C_DIS
LIN {X 0.136,Y -576.681,Z 531.391,A 0.000,B 0.000,C 90.000,E1 106.315} C_DIS
LIN {X -0.290,Y -581.743,Z 531.388,A 0.000,B 0.000,C 90.000,E1 105.843} C_DIS
LIN {X -0.161,Y -586.514,Z 531.385,A 0.000,B 0.000,C 90.000,E1 105.300} C_DIS
LIN {X -0.129,Y -592.653,Z 531.381,A 0.000,B 0.000,C 90.000,E1 104.537} C_DIS
LIN {X 0.058,Y -595.646,Z 531.379,A 0.000,B 0.000,C 90.000,E1 104.120} C_DIS
LIN {X -0.242,Y -597.594,Z 531.377,A 0.000,B 0.000,C 90.000,E1 103.883} C_DIS
LIN {X -0.029,Y -600.387,Z 531.375,A 0.000,B 0.000,C 90.000,E1 103.467} C_DIS
LIN {X 0.270,Y -602.273,Z 531.373,A 0.000,B 0.000,C 90.000,E1 103.175} C_DIS
LIN {X -0.237,Y -606.632,Z 531.370,A 0.000,B 0.000,C 90.000,E1 102.591} C_DIS
LIN {X 0.166,Y -611.750,Z 531.366,A 0.000,B 0.000,C 90.000,E1 101.771} C_DIS
LIN {X -0.180,Y -615.608,Z 531.362,A 0.000,B 0.000,C 90.000,E1 101.186} C_DIS
LIN {X -0.078,Y -619.210,Z 531.359,A 0.000,B 0.000,C 90.000,E1 100.546} C_DIS
LIN {X -0.158,Y -623.267,Z 531.354,A 0.000,B 0.000,C 90.000,E1 99.782} C_DIS
LIN {X 0.004,Y -628.367,Z 531.349,A 0.000,B 0.000,C 90.000,E1 98.746} C_DIS
LIN {X 0.058,Y -631.352,Z 531.345,A 0.000,B 0.000,C 90.000,E1 98.106} C_DIS
LIN {X -0.128,Y -638.139,Z 531.337,A 0.000,B 0.000,C 90.000,E1 96.606} C_DIS
LIN {X -0.137,Y -641.471,Z 531.333,A 0.000,B 0.000,C 90.000,E1 95.853} C_DIS
LIN {X -0.181,Y -644.504,Z 531.328,A 0.000,B 0.000,C 90.000,E1 95.106} C_DIS
LIN {X 0.040,Y -646.438,Z 531.326,A 0.000,B 0.000,C 90.000,E1 94.588} C_DIS
LIN {X 0.226,Y -648.194,Z 531.323,A 0.000,B 0.000,C 90.000,E1 94.073} C_DIS
LIN {X 0.075,Y -651.297,Z 531.317,A 0.000,B 0.000,C 90.000,E1 93.094} C_DIS
LIN {X 0.302,Y -652.652,Z 531.315,A 0.000,B 0.000,C 90.000,E1 92.579} C_DIS
LIN {X -0.310,Y -654.395,Z 531.310,A 0.000,B 0.000,C 90.000,E1 91.892} C_DIS
LIN {X -0.234,Y -655.717,Z 531.306,A 0.000,B 0.000,C 90.000,E1 91.146} C_DIS
LIN {X 0.033,Y -656.352,Z 531.304,A 0.000,B 0.000,C 90.000,E1 90.630} C_DIS
LIN {X 0.304,Y -656.825,Z 531.301,A 0.000,B 0.000,C 90.000,E1 90.115} C_DIS
LIN {X -0.266,Y -657.188,Z 531.297,A 0.000,B 0.000,C 90.000,E1 89.427} C_DIS
LIN {X -0.180,Y -657.183,Z 531.293,A 0.000,B 0.000,C 90.000,E1 88.682} C_DIS
LIN {X 0.286,Y -657.151,Z 531.291,A 0.000,B 0.000,C 90.000,E1 88.396} C_DIS
LIN {X -0.264,Y -656.652,Z 531.287,A 0.000,B 0.000,C 90.000,E1 87.707} C_DIS
LIN {X 0.006,Y -656.197,Z 531.284,A 0.000,B 0.000,C 90.000,E1 87.192} C_DIS
LIN {X 0.108,Y -655.203,Z 531.280,A 0.000,B 0.000,C 90.000,E1 86.445} C_DIS
LIN {X -0.091,Y -654.852,Z 531.279,A 0.000,B 0.000,C 90.000,E1 86.216} C_DIS
LIN {X 0.286,Y -652.232,Z 531.272,A 0.000,B 0.000,C 90.000,E1 84.951} C_DIS
LIN {X -0.298,Y -650.303,Z 531.268,A 0.000,B 0.000,C 90.000,E1 84.261} C_DIS
LIN {X -0.028,Y -648.898,Z 531.265,A 0.000,B 0.000,C 90.000,E1 83.742} C_DIS
LIN {X -0.163,Y -645.732,Z 531.260,A 0.000,B 0.000,C 90.000,E1 82.761} C_DIS
LIN {X -0.087,Y -642.946,Z 531.256,A 0.000,B 0.000,C 90.000,E1 82.008} C_DIS
LIN {X -0.304,Y -638.886,Z 531.250,A 0.000,B 0.000,C 90.000,E1 81.027} C_DIS
LIN {X 0.290,Y -634.914,Z 531.245,A 0.000,B 0.000,C 90.000,E1 80.095} C_DIS
LIN {X -0.222,Y -631.715,Z 531.242,A 0.000,B 0.000,C 90.000,E1 79.511} C_DIS
LIN {X -0.129,Y -628.457,Z 531.238,A 0.000,B 0.000,C 90.000,E1 78.870} C_DIS
LIN {X -0.112,Y -624.344,Z 531.234,A 0.000,B 0.000,C 90.000,E1 78.105} C_DIS
LIN {X -0.270,Y -619.886,Z 531.230,A 0.000,B 0.000,C 90.000,E1 77.353} C_DIS
LIN {X -0.155,Y -616.020,Z 531.226,A 0.000,B 0.000,C 90.000,E1 76.700} C_DIS
LIN {X 0.278,Y -609.743,Z 531.221,A 0.000,B 0.000,C 90.000,E1 75.755} C_DIS
LIN {X 0.152,Y -604.597,Z 531.217,A 0.000,B 0.000,C 90.000,E1 75.117} C_DIS
LIN {X 0.131,Y -598.806,Z 531.214,A 0.000,B 0.000,C 90.000,E1 74.464} C_DIS
LIN {X -0.106,Y -594.071,Z 531.211,A 0.000,B 0.000,C 90.000,E1 73.976} C_DIS
LIN {X -0.264,Y -589.177,Z 531.208,A 0.000,B 0.000,C 90.000,E1 73.504} C_DIS
LIN {X 0.288,Y -583.649,Z 531.206,A 0.000,B 0.000,C 90.000,E1 72.960} C_DIS
LIN {X -0.220,Y -577.901,Z 531.203,A 0.000,B 0.000,C 90.000,E1 72.543} C_DIS
LIN {X 0.230,Y -571.944,Z 531.201,A 0.000,B 0.000,C 90.000,E1 72.054} C_DIS
LIN {X -0.075,Y -567.418,Z 531.199,A 0.000,B 0.000,C 90.000,E1 71.764} C_DIS
LIN {X 0.165,Y -560.796,Z 531.196,A 0.000,B 0.000,C 90.000,E1 71.329} C_DIS
LIN {X 0.233,Y -555.884,Z 531.195,A 0.000,B 0.000,C 90.000,E1 71.040} C_DIS
LIN {X 0.180,Y -550.757,Z 531.193,A 0.000,B 0.000,C 90.000,E1 70.786} C_DIS
LIN {X -0.040,Y -543.944,Z 531.192,A 0.000,B 0.000,C 90.000,E1 70.496} C_DIS
LIN {X 0.171,Y -536.767,Z 531.190,A 0.000,B 0.000,C 90.000,E1 70.188} C_DIS
LIN {X 0.056,Y -531.124,Z 531.189,A 0.000,B 0.000,C 90.000,E1 70.007} C_DIS
LIN {X -0.188,Y -521.885,Z 531.187,A 0.000,B 0.000,C 90.000,E1 69.752} C_DIS
LIN {X -0.135,Y -507.425,Z 531.185,A 0.000,B 0.000,C 90.000,E1 69.337} C_DIS
LIN {X 0.102,Y -496.219,Z 531.184,A 0.000,B 0.000,C 90.000,E1 69.028} C_DIS
LIN {X -0.239,Y -467.732,Z 531.180,A 0.000,B 0.000,C 90.000,E1 68.411} C_DIS
LIN {X 0.150,Y -467.518,Z 531.180,A 0.000,B 0.000,C 90.000,E1 68.358} C_DIS
LIN {X 0.045,Y -465.482,Z 531.172,A 0.000,B 0.000,C 90.000,E1 66.975} C_DIS
LIN {X -0.175,Y -457.042,Z 531.149,A 0.000,B 0.000,C 90.000,E1 62.871} C_DIS
LIN {X -0.066,Y -455.456,Z 531.144,A 0.000,B 0.000,C 90.000,E1 61.897} C_DIS
LIN {X -0.128,Y -446.116,Z 531.121,A 0.000,B 0.000,C 90.000,E1 57.709} C_DIS
LIN {X 0.131,Y -444.435,Z 531.115,A 0.000,B 0.000,C 90.000,E1 56.755} C_DIS
LIN {X 0.092,Y -444.432,Z 531.115,A 0.000,B 0.000,C 90.000,E1 56.755} C_DIS
LIN {X -0.119,Y -448.486,Z 531.106,A 0.000,B 0.000,C 90.000,E1 55.102} C_DIS
LIN {X -0.018,Y -450.614,Z 531.101,A 0.000,B 0.000,C 90.000,E1 54.116} C_DIS
LIN {X -0.178,Y -453.325,Z 531.094,A 0.000,B 0.000,C 90.000,E1 52.844} C_DIS
LIN {X -0.025,Y -455.739,Z 531.086,A 0.000,B 0.000,C 90.000,E1 51.537} C_DIS
LIN {X -0.191,Y -457.892,Z 531.079,A 0.000,B 0.000,C 90.000,E1 50.275} C_DIS
LIN {X -0.087,Y -458.924,Z 531.076,A 0.000,B 0.000,C 90.000,E1 49.622} C_DIS
LIN {X 0.133,Y -461.189,Z 531.067,A 0.000,B 0.000,C 90.000,E1 48.000} C_DIS
LIN {X 0.010,Y -462.662,Z 531.060,A 0.000,B 0.000,C 90.000,E1 46.743} C_DIS
LIN {X -0.149,Y -463.546,Z 531.054,A 0.000,B 0.000,C 90.000,E1 45.810} C_DIS
LIN {X 0.083,Y -464.419,Z 531.047,A 0.000,B 0.000,C 90.000,E1 44.514} C_DIS
LIN {X -0.056,Y -464.905,Z 531.042,A 0.000,B 0.000,C 90.000,E1 43.581} C_DIS
LIN {X 0.131,Y -465.273,Z 531.037,A 0.000,B 0.000,C 90.000,E1 42.609} C_DIS
LIN {X 0.060,Y -465.475,Z 531.030,A 0.000,B 0.000,C 90.000,E1 41.353} C_DIS
LIN {X 0.033,Y -465.414,Z 531.023,A 0.000,B 0.000,C 90.000,E1 40.092} C_DIS
LIN {X -0.231,Y -465.091,Z 531.014,A 0.000,B 0.000,C 90.000,E1 38.543} C_DIS
LIN {X -0.136,Y -464.534,Z 531.005,A 0.000,B 0.000,C 90.000,E1 36.950} C_DIS
LIN {X -0.063,Y -463.810,Z 530.996,A 0.000,B 0.000,C 90.000,E1 35.358} C_DIS
LIN {X -0.027,Y -462.897,Z 530.986,A 0.000,B 0.000,C 90.000,E1 33.452} C_DIS
LIN {X 0.131,Y -461.756,Z 530.974,A 0.000,B 0.000,C 90.000,E1 31.209} C_DIS
LIN {X 0.003,Y -460.446,Z 530.961,A 0.000,B 0.000,C 90.000,E1 28.999} C_DIS
LIN {X 0.078,Y -459.334,Z 530.951,A 0.000,B 0.000,C 90.000,E1 27.078} C_DIS
LIN {X 0.046,Y -458.109,Z 530.938,A 0.000,B 0.000,C 90.000,E1 24.847} C_DIS
LIN {X 0.112,Y -456.989,Z 530.924,A 0.000,B 0.000,C 90.000,E1 22.280} C_DIS
LIN {X -0.208,Y -456.057,Z 530.910,A 0.000,B 0.000,C 90.000,E1 19.758} C_DIS
LIN {X -0.089,Y -455.546,Z 530.899,A 0.000,B 0.000,C 90.000,E1 17.819} C_DIS
LIN {X -0.017,Y -455.281,Z 530.890,A 0.000,B 0.000,C 90.000,E1 16.205} C_DIS
LIN {X -0.098,Y -455.180,Z 530.876,A 0.000,B 0.000,C 90.000,E1 13.647} C_DIS
LIN {X -0.046,Y -455.409,Z 530.865,A 0.000,B 0.000,C 90.000,E1 11.715} C_DIS
LIN {X -0.070,Y -455.858,Z 530.854,A 0.000,B 0.000,C 90.000,E1 9.792} C_DIS
LIN {X 0.070,Y -456.696,Z 530.842,A 0.000,B 0.000,C 90.000,E1 7.530} C_DIS
LIN {X -0.166,Y -458.389,Z 530.824,A 0.000,B 0.000,C 90.000,E1 4.359} C_DIS
LIN {X 0.011,Y -460.726,Z 530.806,A 0.000,B 0.000,C 90.000,E1 1.146} C_DIS
LIN {X -0.161,Y -463.706,Z 530.790,A 0.000,B 0.000,C 90.000,E1 358.224} C_DIS
LIN {X 0.003,Y -466.301,Z 530.778,A 0.000,B 0.000,C 90.000,E1 355.988} C_DIS
LIN {X 0.047,Y -468.736,Z 530.767,A 0.000,B 0.000,C 90.000,E1 354.090} C_DIS
LIN {X 0.199,Y -471.288,Z 530.757,A 0.000,B 0.000,C 90.000,E1 352.186} C_DIS
LIN {X -0.161,Y -474.364,Z 530.745,A 0.000,B 0.000,C 90.000,E1 350.038} C_DIS
LIN {X -0.099,Y -478.486,Z 530.729,A 0.000,B 0.000,C 90.000,E1 347.229} C_DIS
LIN {X -0.117,Y -482.818,Z 530.715,A 0.000,B 0.000,C 90.000,E1 344.755} C_DIS
LIN {X -0.085,Y -487.008,Z 530.703,A 0.000,B 0.000,C 90.000,E1 342.598} C_DIS
LIN {X 0.211,Y -491.243,Z 530.691,A 0.000,B 0.000,C 90.000,E1 340.423} C_DIS
LIN {X 0.230,Y -494.272,Z 530.683,A 0.000,B 0.000,C 90.000,E1 338.901} C_DIS
LIN {X -0.034,Y -496.714,Z 530.676,A 0.000,B 0.000,C 90.000,E1 337.720} C_DIS
LIN {X -0.131,Y -500.283,Z 530.666,A 0.000,B 0.000,C 90.000,E1 335.921} C_DIS
LIN {X 0.040,Y -503.676,Z 530.656,A 0.000,B 0.000,C 90.000,E1 334.101} C_DIS
LIN {X -0.032,Y -506.447,Z 530.648,A 0.000,B 0.000,C 90.000,E1 332.615} C_DIS
LIN {X -0.050,Y -509.222,Z 530.640,A 0.000,B 0.000,C 90.000,E1 331.129} C_DIS
LIN {X 0.127,Y -512.462,Z 530.630,A 0.000,B 0.000,C 90.000,E1 329.331} C_DIS
LIN {X -0.057,Y -515.821,Z 530.620,A 0.000,B 0.000,C 90.000,E1 327.582} C_DIS
LIN {X 0.108,Y -519.201,Z 530.610,A 0.000,B 0.000,C 90.000,E1 325.801} C_DIS
LIN {X -0.039,Y -522.001,Z 530.602,A 0.000,B 0.000,C 90.000,E1 324.356} C_DIS
LIN {X -0.017,Y -525.832,Z 530.591,A 0.000,B 0.000,C 90.000,E1 322.316} C_DIS
LIN {X -0.141,Y -528.086,Z 530.584,A 0.000,B 0.000,C 90.000,E1 321.170} C_DIS
LIN {X -0.045,Y -532.681,Z 530.571,A 0.000,B 0.000,C 90.000,E1 318.852} C_DIS
LIN {X 0.145,Y -536.850,Z 530.560,A 0.000,B 0.000,C 90.000,E1 316.824} C_DIS
LIN {X 0.061,Y -540.512,Z 530.551,A 0.000,B 0.000,C 90.000,E1 315.121} C_DIS
LIN {X 0.066,Y -545.547,Z 530.538,A 0.000,B 0.000,C 90.000,E1 312.852} C_DIS
LIN {X -0.140,Y -550.876,Z 530.526,A 0.000,B 0.000,C 90.000,E1 310.620} C_DIS
LIN {X 0.016,Y -553.346,Z 530.519,A 0.000,B 0.000,C 90.000,E1 309.483} C_DIS
LIN {X -0.073,Y -556.246,Z 530.512,A 0.000,B 0.000,C 90.000,E1 308.096} C_DIS
LIN {X -0.057,Y -560.750,Z 530.500,A 0.000,B 0.000,C 90.000,E1 306.011} C_DIS
LIN {X 0.114,Y -561.824,Z 530.498,A 0.000,B 0.000,C 90.000,E1 305.678} C_DIS
LIN {X 0.099,Y -563.018,Z 530.496,A 0.000,B 0.000,C 90.000,E1 305.264} C_DIS
LIN {X 0.052,Y -564.417,Z 530.494,A 0.000,B 0.000,C 90.000,E1 304.978} C_DIS
LIN {X 0.158,Y -565.432,Z 530.493,A 0.000,B 0.000,C 90.000,E1 304.692} C_DIS
LIN {X 0.053,Y -566.130,Z 530.492,A 0.000,B 0.000,C 90.000,E1 304.565} C_DIS
LIN {X 0.165,Y -567.881,Z 530.491,A 0.000,B 0.000,C 90.000,E1 304.278} C_DIS
LIN {X 0.062,Y -568.558,Z 530.490,A 0.000,B 0.000,C 90.000,E1 304.151} C_DIS
LIN {X -0.070,Y -571.298,Z 530.488,A 0.000,B 0.000,C 90.000,E1 303.754} C_DIS
LIN {X -0.039,Y -578.056,Z 530.482,A 0.000,B 0.000,C 90.000,E1 302.832} C_DIS
